// TIA Portal V20 export
FUNCTION_BLOCK "Sequence_1_WebGuid"   // FB127, LAD
TITLE = Sequence
// Sequence template programmend in ladder logic
// stored: IsIECCheckEnabled true, MemoryReserve 100, Namespace Unit1.Em3, SetENOAutomatically true
   VAR
      instSequenceLADControl { ExternalWritable := 'False'} : "LAF_ControlLadSequence";
      instSequenceLADStatus { ExternalWritable := 'False'} : "LAF_StatusLadSequence";
      statPulse { ExternalWritable := 'False'} : Array[0..999] of Bool;
      statTonTimer { ExternalWritable := 'False'} : Array[0..1099] of TON_TIME;
   END_VAR
   VAR_TEMP
      tempCustomerAction : Bool;   // Placeholder for possible actions
      tempDo_nothing_and_wait_for_init : Bool;   // Placeholder for doing nothing
      tempSafeStateCondition : Bool;   // Temp Condition for the equipment module to be in a safe state
   END_VAR
   VAR CONSTANT
      STEP_IDLE : DInt := 1;   // Idle Step
      JOB_1_STEP_01 : DInt := 101;
      JOB_1_STEP_11 : DInt := 111;
      JOB_1_STEP_21 : DInt := 121;
      JOB_1_STEP_31 : DInt := 131;
      JOB_1_STEP_41 : DInt := 141;
      JOB_1_STEP_51 : DInt := 151;
      JOB_1_STEP_61 : DInt := 161;
      JOB_1_STEP_71 : DInt := 171;
      JOB_1_STEP_81 : DInt := 181;
      JOB_1_STEP_91 : DInt := 191;
      JOB_2_STEP_01 : DInt := 201;
      JOB_2_STEP_11 : DInt := 211;
      JOB_2_STEP_21 : DInt := 221;
      JOB_2_STEP_31 : DInt := 231;
      JOB_2_STEP_41 : DInt := 241;
      JOB_2_STEP_51 : DInt := 251;
      JOB_2_STEP_61 : DInt := 261;
      JOB_2_STEP_71 : DInt := 271;
      JOB_2_STEP_81 : DInt := 281;
      JOB_2_STEP_91 : DInt := 291;
      JOB_3_STEP_01 : DInt := 301;
      JOB_3_STEP_11 : DInt := 311;
      JOB_3_STEP_21 : DInt := 321;
      JOB_3_STEP_31 : DInt := 331;
      JOB_3_STEP_41 : DInt := 341;
      JOB_3_STEP_51 : DInt := 351;
      JOB_3_STEP_61 : DInt := 361;
      JOB_3_STEP_71 : DInt := 371;
      JOB_3_STEP_81 : DInt := 381;
      JOB_3_STEP_91 : DInt := 391;
      JOB_4_STEP_01 : DInt := 401;
      JOB_4_STEP_11 : DInt := 411;
      JOB_4_STEP_21 : DInt := 421;
      JOB_4_STEP_31 : DInt := 431;
      JOB_4_STEP_41 : DInt := 441;
      JOB_4_STEP_51 : DInt := 451;
      JOB_4_STEP_61 : DInt := 461;
      JOB_4_STEP_71 : DInt := 471;
      JOB_4_STEP_81 : DInt := 481;
      JOB_4_STEP_91 : DInt := 491;
      JOB_5_STEP_01 : DInt := 501;
      JOB_5_STEP_11 : DInt := 511;
      JOB_5_STEP_21 : DInt := 521;
      JOB_5_STEP_31 : DInt := 531;
      JOB_5_STEP_41 : DInt := 541;
      JOB_5_STEP_51 : DInt := 551;
      JOB_5_STEP_61 : DInt := 561;
      JOB_5_STEP_71 : DInt := 571;
      JOB_5_STEP_81 : DInt := 581;
      JOB_5_STEP_91 : DInt := 591;
      JOB_6_STEP_01 : DInt := 601;
      JOB_6_STEP_11 : DInt := 611;
      JOB_6_STEP_21 : DInt := 621;
      JOB_6_STEP_31 : DInt := 631;
      JOB_6_STEP_41 : DInt := 641;
      JOB_6_STEP_51 : DInt := 651;
      JOB_6_STEP_61 : DInt := 661;
      JOB_6_STEP_71 : DInt := 671;
      JOB_6_STEP_81 : DInt := 681;
      JOB_6_STEP_91 : DInt := 691;
      JOB_7_STEP_01 : DInt := 701;
      JOB_7_STEP_11 : DInt := 711;
      JOB_7_STEP_21 : DInt := 721;
      JOB_7_STEP_31 : DInt := 731;
      JOB_7_STEP_41 : DInt := 741;
      JOB_7_STEP_51 : DInt := 751;
      JOB_7_STEP_61 : DInt := 761;
      JOB_7_STEP_71 : DInt := 771;
      JOB_7_STEP_81 : DInt := 781;
      JOB_7_STEP_91 : DInt := 791;
      JOB_8_STEP_01 : DInt := 801;
      JOB_8_STEP_11 : DInt := 811;
      JOB_8_STEP_21 : DInt := 821;
      JOB_8_STEP_31 : DInt := 831;
      JOB_8_STEP_41 : DInt := 841;
      JOB_8_STEP_51 : DInt := 851;
      JOB_8_STEP_61 : DInt := 861;
      JOB_8_STEP_71 : DInt := 871;
      JOB_8_STEP_81 : DInt := 881;
      JOB_8_STEP_91 : DInt := 891;
      STEP_IMMEDIATE_STOP : DInt := 901;   // Step executed when an immediate stop command is triggered for the sequence (i.e. when unit is in state aborting)
      TO_DO_INSERT_ACTIONS_HERE : Bool := TRUE;   // Template : Add actions
      TO_DO_INSERT_CONDITION_FOR_TRANSITION_HERE : Bool := TRUE;   // Template : Add conditions
      SeqDelayTime : Time := T#100ms;
      SeqNoDelayTime : Time;
      TRUE : Bool := TRUE;
      FALSE : Bool := FALSE;
   END_VAR
   VAR_TEMP   // added for the SCL form of the ladder/FBD networks
      _w1 : Bool;
      _w2 : Bool;
      _w3 : Bool;
   END_VAR
BEGIN

REGION Network 1: BLOCK INFO HEADER
   // (company) / (C) Copyright (year)
   // ---------------------------------------------------------------------------------
   // Title:                             (Title of this block)
   // Comment/Function: (that is implemented in the block)
   // Library/Family:           (that the source is dedicated to)
   // Author:                        (department / person in charge / contact)
   // Target System:          (test system with FW version)
   // Engineering:              TIA Portal (SW version)
   // Restrictions:               (OB types, etc.)
   // Requirements:           (hardware, technological package, etc.)
   // ---------------------------------------------------------------------------------
   // Change log table:
   // Version          | Date             | Signature      | Expert in charge  | Changes applied ------------------------|----------------------|-------------------------|--------------------------------|-----------------------
   // 001.000.000 | yyyy-mm-dd | 0x00000000 | (name of expert) | First released version
END_REGION

REGION Network 2: DESCRIPTION
   // This is a template block provided by the Automation Framework. It can be used to create an own project.
   // The Block Info Header is prepared to put in your own data.
   // Description of the block could be added here and the docu created by Code2Docu.
END_REGION

REGION Network 3: ******************** CONTROL ********************
END_REGION

REGION Network 4: Sequence Control
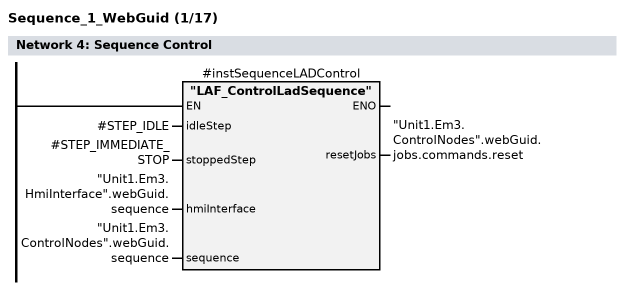
   RUNG wire#powerrail
      #instSequenceLADControl(idleStep := #STEP_IDLE, stoppedStep := #STEP_IMMEDIATE_STOP, hmiInterface := "Unit1.Em3.HmiInterface".webGuid.sequence, sequence := "Unit1.Em3.ControlNodes".webGuid.sequence, resetJobs => "Unit1.Em3.ControlNodes".webGuid.jobs.commands.reset)
   END_RUNG
   // the same network as SCL:
   #instSequenceLADControl(idleStep := #STEP_IDLE,   // "LAF_ControlLadSequence"
                           stoppedStep := #STEP_IMMEDIATE_STOP,
                           hmiInterface := "Unit1.Em3.HmiInterface".webGuid.sequence,
                           sequence := "Unit1.Em3.ControlNodes".webGuid.sequence,
                           resetJobs => "Unit1.Em3.ControlNodes".webGuid.jobs.commands.reset);
END_REGION

REGION Network 5: Step IDLE
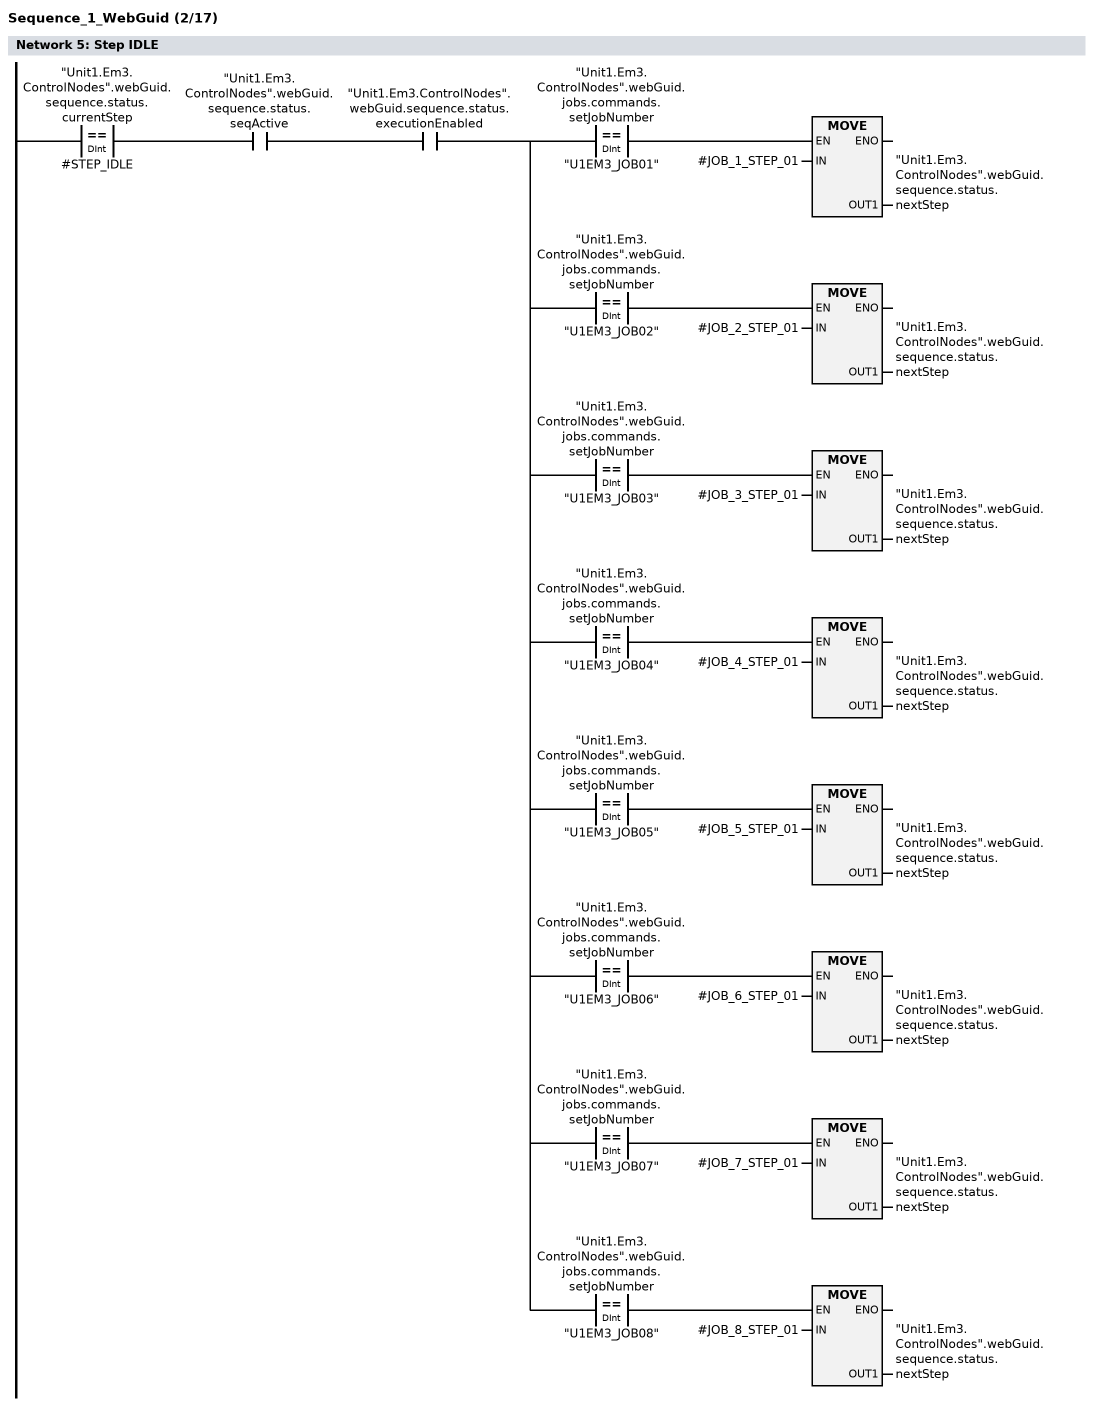
   RUNG wire#powerrail
      { S7_Templates := "SrcType := DInt" } EQ_Contact(in1 := "Unit1.Em3.ControlNodes".webGuid.sequence.status.currentStep, in2 := #STEP_IDLE)
      Contact( "Unit1.Em3.ControlNodes".webGuid.sequence.status.seqActive )
      Contact( "Unit1.Em3.ControlNodes".webGuid.sequence.status.executionEnabled )
      wire#w1
      { S7_Templates := "SrcType := DInt" } EQ_Contact(in1 := "Unit1.Em3.ControlNodes".webGuid.jobs.commands.setJobNumber, in2 := "U1EM3_JOB01")
      Move(in := #JOB_1_STEP_01, out1 => "Unit1.Em3.ControlNodes".webGuid.sequence.status.nextStep)
   END_RUNG
   RUNG wire#w1
      { S7_Templates := "SrcType := DInt" } EQ_Contact(in1 := "Unit1.Em3.ControlNodes".webGuid.jobs.commands.setJobNumber, in2 := "U1EM3_JOB02")
      Move(in := #JOB_2_STEP_01, out1 => "Unit1.Em3.ControlNodes".webGuid.sequence.status.nextStep)
   END_RUNG
   RUNG wire#w1
      { S7_Templates := "SrcType := DInt" } EQ_Contact(in1 := "Unit1.Em3.ControlNodes".webGuid.jobs.commands.setJobNumber, in2 := "U1EM3_JOB03")
      Move(in := #JOB_3_STEP_01, out1 => "Unit1.Em3.ControlNodes".webGuid.sequence.status.nextStep)
   END_RUNG
   RUNG wire#w1
      { S7_Templates := "SrcType := DInt" } EQ_Contact(in1 := "Unit1.Em3.ControlNodes".webGuid.jobs.commands.setJobNumber, in2 := "U1EM3_JOB04")
      Move(in := #JOB_4_STEP_01, out1 => "Unit1.Em3.ControlNodes".webGuid.sequence.status.nextStep)
   END_RUNG
   RUNG wire#w1
      { S7_Templates := "SrcType := DInt" } EQ_Contact(in1 := "Unit1.Em3.ControlNodes".webGuid.jobs.commands.setJobNumber, in2 := "U1EM3_JOB05")
      Move(in := #JOB_5_STEP_01, out1 => "Unit1.Em3.ControlNodes".webGuid.sequence.status.nextStep)
   END_RUNG
   RUNG wire#w1
      { S7_Templates := "SrcType := DInt" } EQ_Contact(in1 := "Unit1.Em3.ControlNodes".webGuid.jobs.commands.setJobNumber, in2 := "U1EM3_JOB06")
      Move(in := #JOB_6_STEP_01, out1 => "Unit1.Em3.ControlNodes".webGuid.sequence.status.nextStep)
   END_RUNG
   RUNG wire#w1
      { S7_Templates := "SrcType := DInt" } EQ_Contact(in1 := "Unit1.Em3.ControlNodes".webGuid.jobs.commands.setJobNumber, in2 := "U1EM3_JOB07")
      Move(in := #JOB_7_STEP_01, out1 => "Unit1.Em3.ControlNodes".webGuid.sequence.status.nextStep)
   END_RUNG
   RUNG wire#w1
      { S7_Templates := "SrcType := DInt" } EQ_Contact(in1 := "Unit1.Em3.ControlNodes".webGuid.jobs.commands.setJobNumber, in2 := "U1EM3_JOB08")
      Move(in := #JOB_8_STEP_01, out1 => "Unit1.Em3.ControlNodes".webGuid.sequence.status.nextStep)
   END_RUNG
   // the same network as SCL:
   #_w1 := ("Unit1.Em3.ControlNodes".webGuid.sequence.status.currentStep = #STEP_IDLE) AND "Unit1.Em3.ControlNodes".webGuid.sequence.status.seqActive AND "Unit1.Em3.ControlNodes".webGuid.sequence.status.executionEnabled;
   IF #_w1 AND ("Unit1.Em3.ControlNodes".webGuid.jobs.commands.setJobNumber = "U1EM3_JOB01") THEN
       "Unit1.Em3.ControlNodes".webGuid.sequence.status.nextStep := #JOB_1_STEP_01;
   END_IF;
   IF #_w1 AND ("Unit1.Em3.ControlNodes".webGuid.jobs.commands.setJobNumber = "U1EM3_JOB02") THEN
       "Unit1.Em3.ControlNodes".webGuid.sequence.status.nextStep := #JOB_2_STEP_01;
   END_IF;
   IF #_w1 AND ("Unit1.Em3.ControlNodes".webGuid.jobs.commands.setJobNumber = "U1EM3_JOB03") THEN
       "Unit1.Em3.ControlNodes".webGuid.sequence.status.nextStep := #JOB_3_STEP_01;
   END_IF;
   IF #_w1 AND ("Unit1.Em3.ControlNodes".webGuid.jobs.commands.setJobNumber = "U1EM3_JOB04") THEN
       "Unit1.Em3.ControlNodes".webGuid.sequence.status.nextStep := #JOB_4_STEP_01;
   END_IF;
   IF #_w1 AND ("Unit1.Em3.ControlNodes".webGuid.jobs.commands.setJobNumber = "U1EM3_JOB05") THEN
       "Unit1.Em3.ControlNodes".webGuid.sequence.status.nextStep := #JOB_5_STEP_01;
   END_IF;
   IF #_w1 AND ("Unit1.Em3.ControlNodes".webGuid.jobs.commands.setJobNumber = "U1EM3_JOB06") THEN
       "Unit1.Em3.ControlNodes".webGuid.sequence.status.nextStep := #JOB_6_STEP_01;
   END_IF;
   IF #_w1 AND ("Unit1.Em3.ControlNodes".webGuid.jobs.commands.setJobNumber = "U1EM3_JOB07") THEN
       "Unit1.Em3.ControlNodes".webGuid.sequence.status.nextStep := #JOB_7_STEP_01;
   END_IF;
   IF #_w1 AND ("Unit1.Em3.ControlNodes".webGuid.jobs.commands.setJobNumber = "U1EM3_JOB08") THEN
       "Unit1.Em3.ControlNodes".webGuid.sequence.status.nextStep := #JOB_8_STEP_01;
   END_IF;
END_REGION

REGION Network 6: Step IDLE Dancer WorkPos Command
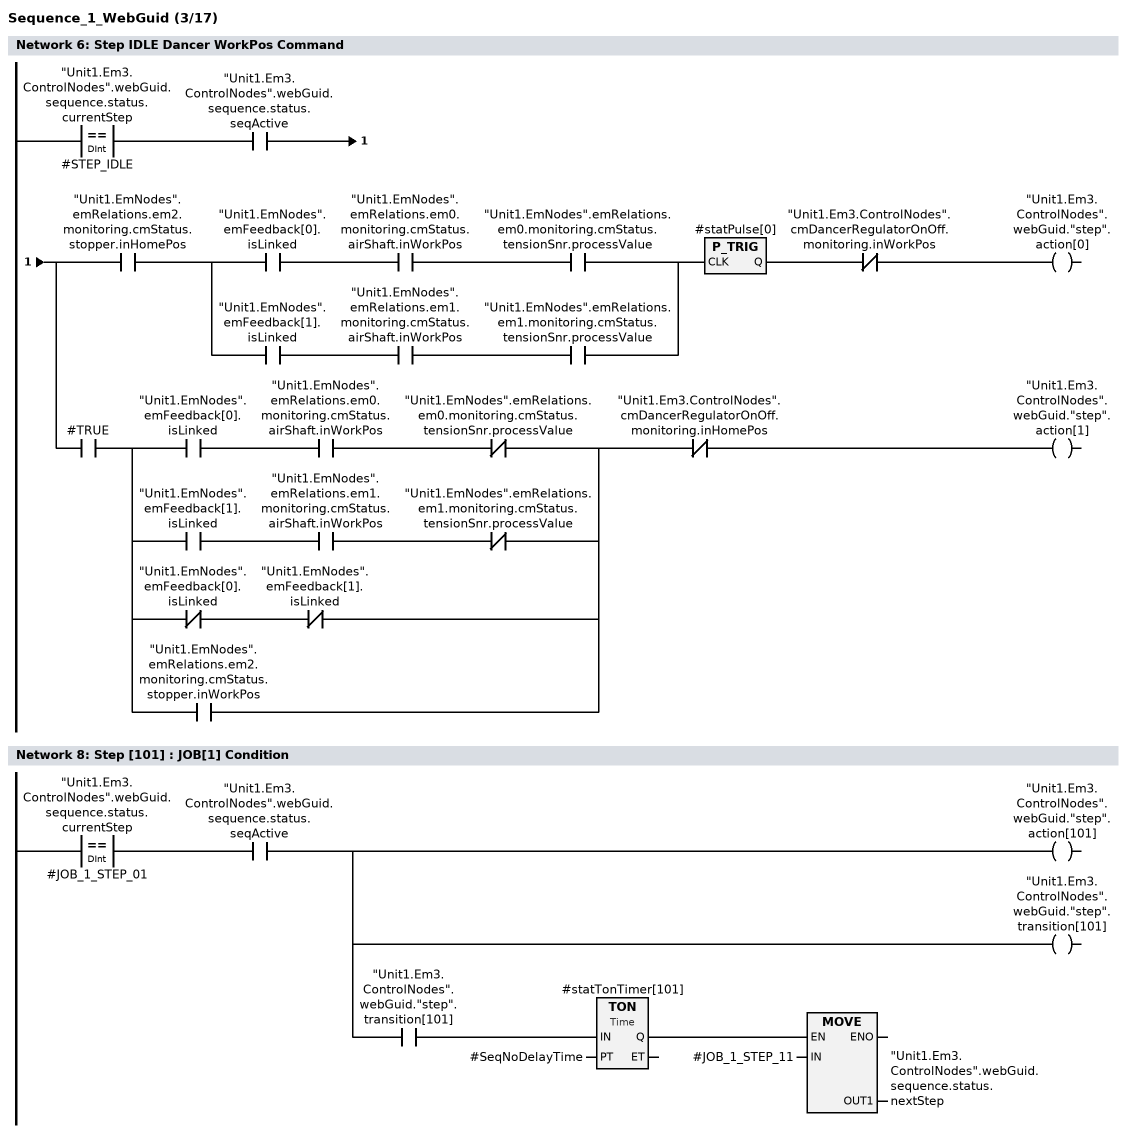
   RUNG wire#powerrail
      { S7_Templates := "SrcType := DInt" } EQ_Contact(in1 := "Unit1.Em3.ControlNodes".webGuid.sequence.status.currentStep, in2 := #STEP_IDLE)
      Contact( "Unit1.Em3.ControlNodes".webGuid.sequence.status.seqActive )
      wire#w1
      Contact( "Unit1.EmNodes".emRelations.em2.monitoring.cmStatus.stopper.inHomePos )
      wire#w2
      Contact( "Unit1.EmNodes".emFeedback[0].isLinked )
      Contact( "Unit1.EmNodes".emRelations.em0.monitoring.cmStatus.airShaft.inWorkPos )
      Contact( "Unit1.EmNodes".emRelations.em0.monitoring.cmStatus.tensionSnr.processValue )
      wire#w3
      P_Trig( #statPulse[0] )
      I_Contact( "Unit1.Em3.ControlNodes".cmDancerRegulatorOnOff.monitoring.inWorkPos )
      Coil( "Unit1.Em3.ControlNodes".webGuid."step".action[0] )
   END_RUNG
   RUNG wire#w2
      Contact( "Unit1.EmNodes".emFeedback[1].isLinked )
      Contact( "Unit1.EmNodes".emRelations.em1.monitoring.cmStatus.airShaft.inWorkPos )
      Contact( "Unit1.EmNodes".emRelations.em1.monitoring.cmStatus.tensionSnr.processValue )
   END_RUNG wire#w3
   RUNG wire#w1
      Contact( #TRUE )
      wire#w4
      Contact( "Unit1.EmNodes".emFeedback[0].isLinked )
      Contact( "Unit1.EmNodes".emRelations.em0.monitoring.cmStatus.airShaft.inWorkPos )
      I_Contact( "Unit1.EmNodes".emRelations.em0.monitoring.cmStatus.tensionSnr.processValue )
      wire#w5
      I_Contact( "Unit1.Em3.ControlNodes".cmDancerRegulatorOnOff.monitoring.inHomePos )
      Coil( "Unit1.Em3.ControlNodes".webGuid."step".action[1] )
   END_RUNG
   RUNG wire#w4
      Contact( "Unit1.EmNodes".emFeedback[1].isLinked )
      Contact( "Unit1.EmNodes".emRelations.em1.monitoring.cmStatus.airShaft.inWorkPos )
      I_Contact( "Unit1.EmNodes".emRelations.em1.monitoring.cmStatus.tensionSnr.processValue )
   END_RUNG wire#w5
   RUNG wire#w4
      I_Contact( "Unit1.EmNodes".emFeedback[0].isLinked )
      I_Contact( "Unit1.EmNodes".emFeedback[1].isLinked )
   END_RUNG wire#w5
   RUNG wire#w4
      Contact( "Unit1.EmNodes".emRelations.em2.monitoring.cmStatus.stopper.inWorkPos )
   END_RUNG wire#w5
   // the same network as SCL:
   #_w1 := ("Unit1.Em3.ControlNodes".webGuid.sequence.status.currentStep = #STEP_IDLE) AND "Unit1.Em3.ControlNodes".webGuid.sequence.status.seqActive;
   #_w2 := #_w1 AND "Unit1.EmNodes".emRelations.em2.monitoring.cmStatus.stopper.inHomePos AND (("Unit1.EmNodes".emFeedback[0].isLinked AND "Unit1.EmNodes".emRelations.em0.monitoring.cmStatus.airShaft.inWorkPos AND "Unit1.EmNodes".emRelations.em0.monitoring.cmStatus.tensionSnr.processValue) OR ("Unit1.EmNodes".emFeedback[1].isLinked AND "Unit1.EmNodes".emRelations.em1.monitoring.cmStatus.airShaft.inWorkPos AND "Unit1.EmNodes".emRelations.em1.monitoring.cmStatus.tensionSnr.processValue));
   #_w3 := #_w2 AND NOT #statPulse[0];   // rising edge
   #statPulse[0] := #_w2;
   "Unit1.Em3.ControlNodes".webGuid."step".action[0] := #_w3 AND NOT "Unit1.Em3.ControlNodes".cmDancerRegulatorOnOff.monitoring.inWorkPos;
   "Unit1.Em3.ControlNodes".webGuid."step".action[1] := #_w1 AND #TRUE AND (("Unit1.EmNodes".emFeedback[0].isLinked AND "Unit1.EmNodes".emRelations.em0.monitoring.cmStatus.airShaft.inWorkPos AND NOT "Unit1.EmNodes".emRelations.em0.monitoring.cmStatus.tensionSnr.processValue) OR ("Unit1.EmNodes".emFeedback[1].isLinked AND "Unit1.EmNodes".emRelations.em1.monitoring.cmStatus.airShaft.inWorkPos AND NOT "Unit1.EmNodes".emRelations.em1.monitoring.cmStatus.tensionSnr.processValue) OR (NOT "Unit1.EmNodes".emFeedback[0].isLinked AND NOT "Unit1.EmNodes".emFeedback[1].isLinked) OR "Unit1.EmNodes".emRelations.em2.monitoring.cmStatus.stopper.inWorkPos) AND NOT "Unit1.Em3.ControlNodes".cmDancerRegulatorOnOff.monitoring.inHomePos;
END_REGION

REGION Network 7: ******************** JOB[1] EM INITIALIZED ********************
END_REGION

REGION Network 8: Step [101] : JOB[1] Condition
   RUNG wire#powerrail
      { S7_Templates := "SrcType := DInt" } EQ_Contact(in1 := "Unit1.Em3.ControlNodes".webGuid.sequence.status.currentStep, in2 := #JOB_1_STEP_01)
      Contact( "Unit1.Em3.ControlNodes".webGuid.sequence.status.seqActive )
      wire#w1
      Coil( "Unit1.Em3.ControlNodes".webGuid."step".action[101] )
   END_RUNG
   RUNG wire#w1
      Coil( "Unit1.Em3.ControlNodes".webGuid."step".transition[101] )
   END_RUNG
   RUNG wire#w1
      Contact( "Unit1.Em3.ControlNodes".webGuid."step".transition[101] )
      { S7_Templates := "time_type := Time" } #statTonTimer[101].TON(pt := #SeqNoDelayTime, et =>)
      Move(in := #JOB_1_STEP_11, out1 => "Unit1.Em3.ControlNodes".webGuid.sequence.status.nextStep)
   END_RUNG
   // the same network as SCL:
   "Unit1.Em3.ControlNodes".webGuid."step".action[101] := ("Unit1.Em3.ControlNodes".webGuid.sequence.status.currentStep = #JOB_1_STEP_01) AND "Unit1.Em3.ControlNodes".webGuid.sequence.status.seqActive;
   "Unit1.Em3.ControlNodes".webGuid."step".transition[101] := ("Unit1.Em3.ControlNodes".webGuid.sequence.status.currentStep = #JOB_1_STEP_01) AND "Unit1.Em3.ControlNodes".webGuid.sequence.status.seqActive;
   #statTonTimer[101].TON(IN := ("Unit1.Em3.ControlNodes".webGuid.sequence.status.currentStep = #JOB_1_STEP_01) AND "Unit1.Em3.ControlNodes".webGuid.sequence.status.seqActive AND "Unit1.Em3.ControlNodes".webGuid."step".transition[101],
                          PT := #SeqNoDelayTime);
   IF #statTonTimer[101].Q THEN
       "Unit1.Em3.ControlNodes".webGuid.sequence.status.nextStep := #JOB_1_STEP_11;
   END_IF;
END_REGION

REGION Network 9: Step [111] : Web Guide EPC Mode Check
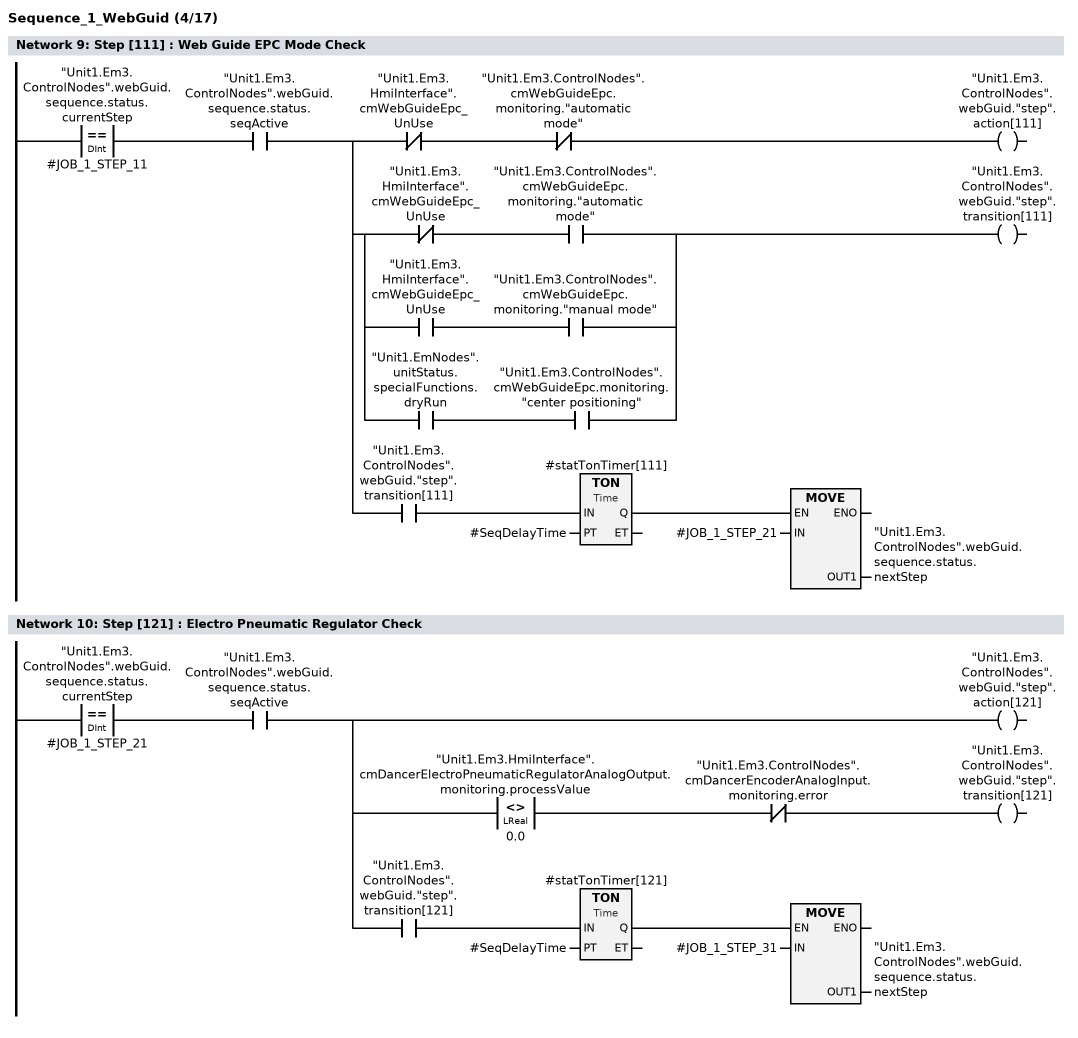
   RUNG wire#powerrail
      { S7_Templates := "SrcType := DInt" } EQ_Contact(in1 := "Unit1.Em3.ControlNodes".webGuid.sequence.status.currentStep, in2 := #JOB_1_STEP_11)
      Contact( "Unit1.Em3.ControlNodes".webGuid.sequence.status.seqActive )
      wire#w1
      I_Contact( "Unit1.Em3.HmiInterface".cmWebGuideEpc_UnUse )
      I_Contact( "Unit1.Em3.ControlNodes".cmWebGuideEpc.monitoring."automatic mode" )
      Coil( "Unit1.Em3.ControlNodes".webGuid."step".action[111] )
   END_RUNG
   RUNG wire#w1
      I_Contact( "Unit1.Em3.HmiInterface".cmWebGuideEpc_UnUse )
      Contact( "Unit1.Em3.ControlNodes".cmWebGuideEpc.monitoring."automatic mode" )
      wire#w2
      Coil( "Unit1.Em3.ControlNodes".webGuid."step".transition[111] )
   END_RUNG
   RUNG wire#w1
      Contact( "Unit1.Em3.HmiInterface".cmWebGuideEpc_UnUse )
      Contact( "Unit1.Em3.ControlNodes".cmWebGuideEpc.monitoring."manual mode" )
   END_RUNG wire#w2
   RUNG wire#w1
      Contact( "Unit1.EmNodes".unitStatus.specialFunctions.dryRun )
      Contact( "Unit1.Em3.ControlNodes".cmWebGuideEpc.monitoring."center positioning" )
   END_RUNG wire#w2
   RUNG wire#w1
      Contact( "Unit1.Em3.ControlNodes".webGuid."step".transition[111] )
      { S7_Templates := "time_type := Time" } #statTonTimer[111].TON(pt := #SeqDelayTime, et =>)
      Move(in := #JOB_1_STEP_21, out1 => "Unit1.Em3.ControlNodes".webGuid.sequence.status.nextStep)
   END_RUNG
   // the same network as SCL:
   #_w1 := ("Unit1.Em3.ControlNodes".webGuid.sequence.status.currentStep = #JOB_1_STEP_11) AND "Unit1.Em3.ControlNodes".webGuid.sequence.status.seqActive;
   "Unit1.Em3.ControlNodes".webGuid."step".action[111] := #_w1 AND NOT "Unit1.Em3.HmiInterface".cmWebGuideEpc_UnUse AND NOT "Unit1.Em3.ControlNodes".cmWebGuideEpc.monitoring."automatic mode";
   "Unit1.Em3.ControlNodes".webGuid."step".transition[111] := #_w1 AND ((NOT "Unit1.Em3.HmiInterface".cmWebGuideEpc_UnUse AND "Unit1.Em3.ControlNodes".cmWebGuideEpc.monitoring."automatic mode") OR ("Unit1.Em3.HmiInterface".cmWebGuideEpc_UnUse AND "Unit1.Em3.ControlNodes".cmWebGuideEpc.monitoring."manual mode") OR ("Unit1.EmNodes".unitStatus.specialFunctions.dryRun AND "Unit1.Em3.ControlNodes".cmWebGuideEpc.monitoring."center positioning"));
   #statTonTimer[111].TON(IN := #_w1 AND "Unit1.Em3.ControlNodes".webGuid."step".transition[111],
                          PT := #SeqDelayTime);
   IF #statTonTimer[111].Q THEN
       "Unit1.Em3.ControlNodes".webGuid.sequence.status.nextStep := #JOB_1_STEP_21;
   END_IF;
END_REGION

REGION Network 10: Step [121] : Electro Pneumatic Regulator Check
   RUNG wire#powerrail
      { S7_Templates := "SrcType := DInt" } EQ_Contact(in1 := "Unit1.Em3.ControlNodes".webGuid.sequence.status.currentStep, in2 := #JOB_1_STEP_21)
      Contact( "Unit1.Em3.ControlNodes".webGuid.sequence.status.seqActive )
      wire#w1
      Coil( "Unit1.Em3.ControlNodes".webGuid."step".action[121] )
   END_RUNG
   RUNG wire#w1
      { S7_Templates := "SrcType := LReal" } NE_Contact(in1 := "Unit1.Em3.HmiInterface".cmDancerElectroPneumaticRegulatorAnalogOutput.monitoring.processValue, in2 := 0.0)
      I_Contact( "Unit1.Em3.ControlNodes".cmDancerEncoderAnalogInput.monitoring.error )
      Coil( "Unit1.Em3.ControlNodes".webGuid."step".transition[121] )
   END_RUNG
   RUNG wire#w1
      Contact( "Unit1.Em3.ControlNodes".webGuid."step".transition[121] )
      { S7_Templates := "time_type := Time" } #statTonTimer[121].TON(pt := #SeqDelayTime, et =>)
      Move(in := #JOB_1_STEP_31, out1 => "Unit1.Em3.ControlNodes".webGuid.sequence.status.nextStep)
   END_RUNG
   // the same network as SCL:
   "Unit1.Em3.ControlNodes".webGuid."step".action[121] := ("Unit1.Em3.ControlNodes".webGuid.sequence.status.currentStep = #JOB_1_STEP_21) AND "Unit1.Em3.ControlNodes".webGuid.sequence.status.seqActive;
   "Unit1.Em3.ControlNodes".webGuid."step".transition[121] := ("Unit1.Em3.ControlNodes".webGuid.sequence.status.currentStep = #JOB_1_STEP_21) AND "Unit1.Em3.ControlNodes".webGuid.sequence.status.seqActive AND ("Unit1.Em3.HmiInterface".cmDancerElectroPneumaticRegulatorAnalogOutput.monitoring.processValue <> 0.0) AND NOT "Unit1.Em3.ControlNodes".cmDancerEncoderAnalogInput.monitoring.error;
   #statTonTimer[121].TON(IN := ("Unit1.Em3.ControlNodes".webGuid.sequence.status.currentStep = #JOB_1_STEP_21) AND "Unit1.Em3.ControlNodes".webGuid.sequence.status.seqActive AND "Unit1.Em3.ControlNodes".webGuid."step".transition[121],
                          PT := #SeqDelayTime);
   IF #statTonTimer[121].Q THEN
       "Unit1.Em3.ControlNodes".webGuid.sequence.status.nextStep := #JOB_1_STEP_31;
   END_IF;
END_REGION

REGION Network 11: Step [131] : Dancer WorkPos Command
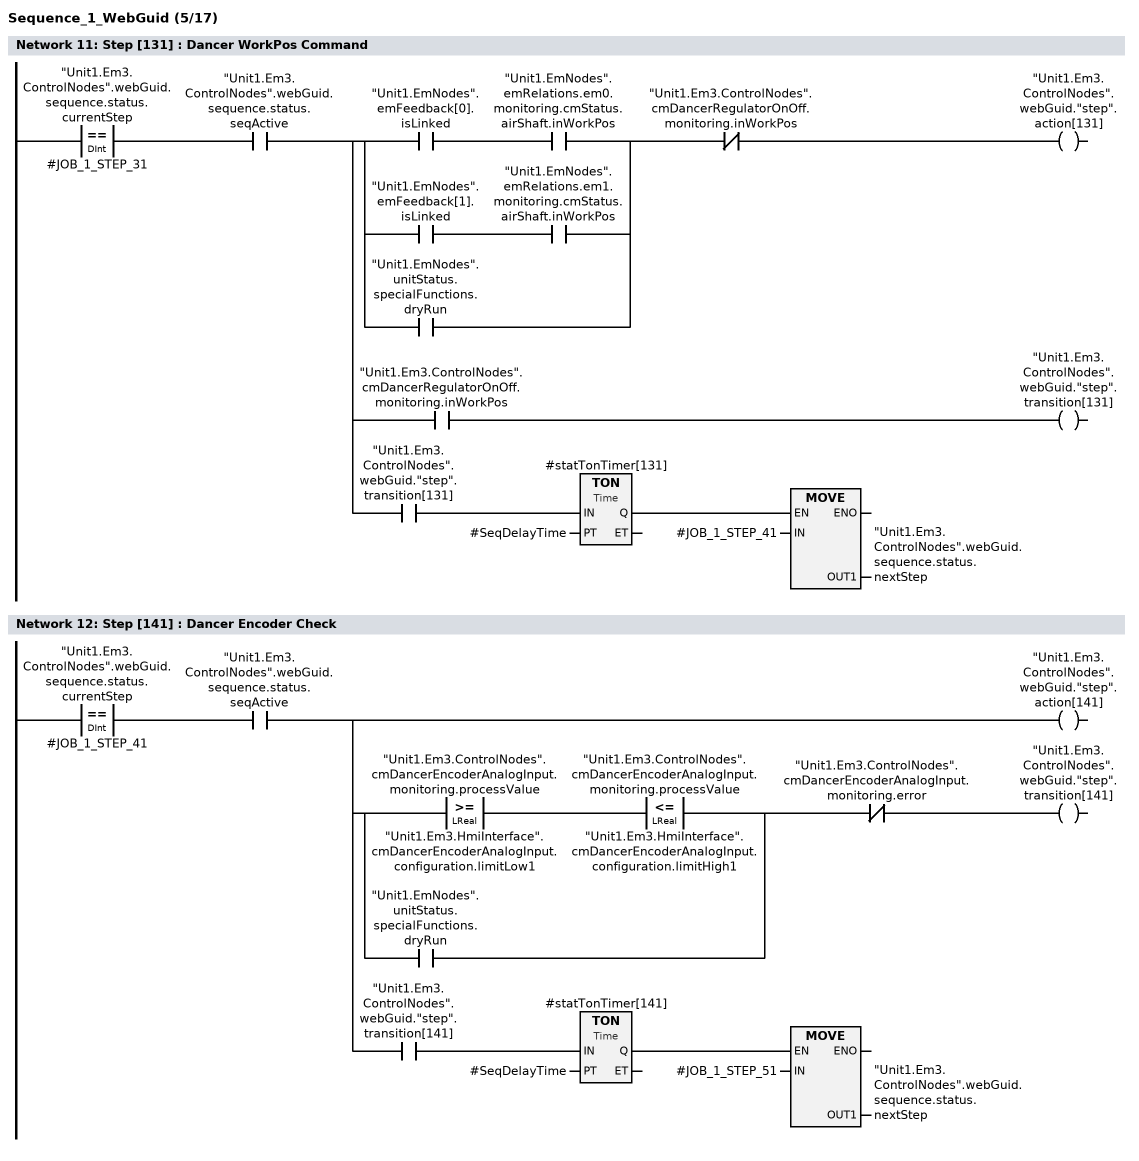
   RUNG wire#powerrail
      { S7_Templates := "SrcType := DInt" } EQ_Contact(in1 := "Unit1.Em3.ControlNodes".webGuid.sequence.status.currentStep, in2 := #JOB_1_STEP_31)
      Contact( "Unit1.Em3.ControlNodes".webGuid.sequence.status.seqActive )
      wire#w1
      Contact( "Unit1.EmNodes".emFeedback[0].isLinked )
      Contact( "Unit1.EmNodes".emRelations.em0.monitoring.cmStatus.airShaft.inWorkPos )
      wire#w2
      I_Contact( "Unit1.Em3.ControlNodes".cmDancerRegulatorOnOff.monitoring.inWorkPos )
      Coil( "Unit1.Em3.ControlNodes".webGuid."step".action[131] )
   END_RUNG
   RUNG wire#w1
      Contact( "Unit1.EmNodes".emFeedback[1].isLinked )
      Contact( "Unit1.EmNodes".emRelations.em1.monitoring.cmStatus.airShaft.inWorkPos )
   END_RUNG wire#w2
   RUNG wire#w1
      Contact( "Unit1.EmNodes".unitStatus.specialFunctions.dryRun )
   END_RUNG wire#w2
   RUNG wire#w1
      Contact( "Unit1.Em3.ControlNodes".cmDancerRegulatorOnOff.monitoring.inWorkPos )
      Coil( "Unit1.Em3.ControlNodes".webGuid."step".transition[131] )
   END_RUNG
   RUNG wire#w1
      Contact( "Unit1.Em3.ControlNodes".webGuid."step".transition[131] )
      { S7_Templates := "time_type := Time" } #statTonTimer[131].TON(pt := #SeqDelayTime, et =>)
      Move(in := #JOB_1_STEP_41, out1 => "Unit1.Em3.ControlNodes".webGuid.sequence.status.nextStep)
   END_RUNG
   // the same network as SCL:
   #_w1 := ("Unit1.Em3.ControlNodes".webGuid.sequence.status.currentStep = #JOB_1_STEP_31) AND "Unit1.Em3.ControlNodes".webGuid.sequence.status.seqActive;
   "Unit1.Em3.ControlNodes".webGuid."step".action[131] := #_w1 AND (("Unit1.EmNodes".emFeedback[0].isLinked AND "Unit1.EmNodes".emRelations.em0.monitoring.cmStatus.airShaft.inWorkPos) OR ("Unit1.EmNodes".emFeedback[1].isLinked AND "Unit1.EmNodes".emRelations.em1.monitoring.cmStatus.airShaft.inWorkPos) OR "Unit1.EmNodes".unitStatus.specialFunctions.dryRun) AND NOT "Unit1.Em3.ControlNodes".cmDancerRegulatorOnOff.monitoring.inWorkPos;
   "Unit1.Em3.ControlNodes".webGuid."step".transition[131] := #_w1 AND "Unit1.Em3.ControlNodes".cmDancerRegulatorOnOff.monitoring.inWorkPos;
   #statTonTimer[131].TON(IN := #_w1 AND "Unit1.Em3.ControlNodes".webGuid."step".transition[131],
                          PT := #SeqDelayTime);
   IF #statTonTimer[131].Q THEN
       "Unit1.Em3.ControlNodes".webGuid.sequence.status.nextStep := #JOB_1_STEP_41;
   END_IF;
END_REGION

REGION Network 12: Step [141] : Dancer Encoder Check
   RUNG wire#powerrail
      { S7_Templates := "SrcType := DInt" } EQ_Contact(in1 := "Unit1.Em3.ControlNodes".webGuid.sequence.status.currentStep, in2 := #JOB_1_STEP_41)
      Contact( "Unit1.Em3.ControlNodes".webGuid.sequence.status.seqActive )
      wire#w1
      Coil( "Unit1.Em3.ControlNodes".webGuid."step".action[141] )
   END_RUNG
   RUNG wire#w1
      { S7_Templates := "SrcType := LReal" } GE_Contact(in1 := "Unit1.Em3.ControlNodes".cmDancerEncoderAnalogInput.monitoring.processValue, in2 := "Unit1.Em3.HmiInterface".cmDancerEncoderAnalogInput.configuration.limitLow1)
      { S7_Templates := "SrcType := LReal" } LE_Contact(in1 := "Unit1.Em3.ControlNodes".cmDancerEncoderAnalogInput.monitoring.processValue, in2 := "Unit1.Em3.HmiInterface".cmDancerEncoderAnalogInput.configuration.limitHigh1)
      wire#w2
      I_Contact( "Unit1.Em3.ControlNodes".cmDancerEncoderAnalogInput.monitoring.error )
      Coil( "Unit1.Em3.ControlNodes".webGuid."step".transition[141] )
   END_RUNG
   RUNG wire#w1
      Contact( "Unit1.EmNodes".unitStatus.specialFunctions.dryRun )
   END_RUNG wire#w2
   RUNG wire#w1
      Contact( "Unit1.Em3.ControlNodes".webGuid."step".transition[141] )
      { S7_Templates := "time_type := Time" } #statTonTimer[141].TON(pt := #SeqDelayTime, et =>)
      Move(in := #JOB_1_STEP_51, out1 => "Unit1.Em3.ControlNodes".webGuid.sequence.status.nextStep)
   END_RUNG
   // the same network as SCL:
   "Unit1.Em3.ControlNodes".webGuid."step".action[141] := ("Unit1.Em3.ControlNodes".webGuid.sequence.status.currentStep = #JOB_1_STEP_41) AND "Unit1.Em3.ControlNodes".webGuid.sequence.status.seqActive;
   "Unit1.Em3.ControlNodes".webGuid."step".transition[141] := ("Unit1.Em3.ControlNodes".webGuid.sequence.status.currentStep = #JOB_1_STEP_41) AND "Unit1.Em3.ControlNodes".webGuid.sequence.status.seqActive AND ((("Unit1.Em3.ControlNodes".cmDancerEncoderAnalogInput.monitoring.processValue >= "Unit1.Em3.HmiInterface".cmDancerEncoderAnalogInput.configuration.limitLow1) AND ("Unit1.Em3.ControlNodes".cmDancerEncoderAnalogInput.monitoring.processValue <= "Unit1.Em3.HmiInterface".cmDancerEncoderAnalogInput.configuration.limitHigh1)) OR "Unit1.EmNodes".unitStatus.specialFunctions.dryRun) AND NOT "Unit1.Em3.ControlNodes".cmDancerEncoderAnalogInput.monitoring.error;
   #statTonTimer[141].TON(IN := ("Unit1.Em3.ControlNodes".webGuid.sequence.status.currentStep = #JOB_1_STEP_41) AND "Unit1.Em3.ControlNodes".webGuid.sequence.status.seqActive AND "Unit1.Em3.ControlNodes".webGuid."step".transition[141],
                          PT := #SeqDelayTime);
   IF #statTonTimer[141].Q THEN
       "Unit1.Em3.ControlNodes".webGuid.sequence.status.nextStep := #JOB_1_STEP_51;
   END_IF;
END_REGION

REGION Network 13: Step [151] : Master Virtual Axis Homed Check
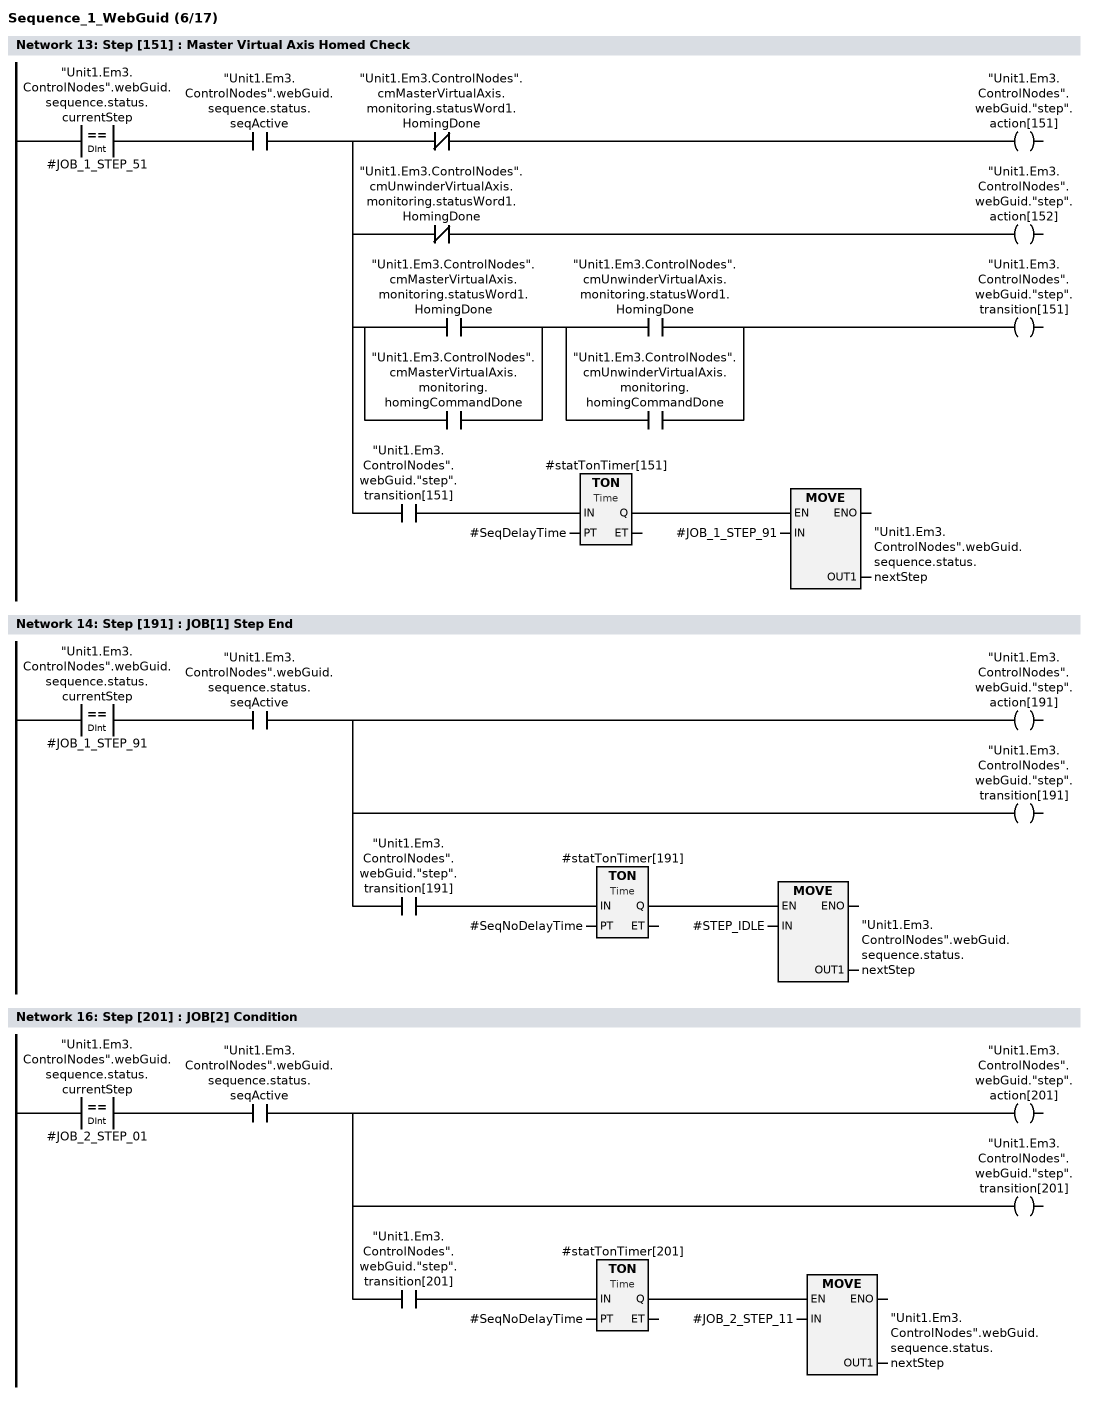
   RUNG wire#powerrail
      { S7_Templates := "SrcType := DInt" } EQ_Contact(in1 := "Unit1.Em3.ControlNodes".webGuid.sequence.status.currentStep, in2 := #JOB_1_STEP_51)
      Contact( "Unit1.Em3.ControlNodes".webGuid.sequence.status.seqActive )
      wire#w1
      I_Contact( "Unit1.Em3.ControlNodes".cmMasterVirtualAxis.monitoring.statusWord1.HomingDone )
      Coil( "Unit1.Em3.ControlNodes".webGuid."step".action[151] )
   END_RUNG
   RUNG wire#w1
      I_Contact( "Unit1.Em3.ControlNodes".cmUnwinderVirtualAxis.monitoring.statusWord1.HomingDone )
      Coil( "Unit1.Em3.ControlNodes".webGuid."step".action[152] )
   END_RUNG
   RUNG wire#w1
      Contact( "Unit1.Em3.ControlNodes".cmMasterVirtualAxis.monitoring.statusWord1.HomingDone )
      wire#w2
      Contact( "Unit1.Em3.ControlNodes".cmUnwinderVirtualAxis.monitoring.statusWord1.HomingDone )
      wire#w3
      Coil( "Unit1.Em3.ControlNodes".webGuid."step".transition[151] )
   END_RUNG
   RUNG wire#w1
      Contact( "Unit1.Em3.ControlNodes".cmMasterVirtualAxis.monitoring.homingCommandDone )
   END_RUNG wire#w2
   RUNG wire#w2
      Contact( "Unit1.Em3.ControlNodes".cmUnwinderVirtualAxis.monitoring.homingCommandDone )
   END_RUNG wire#w3
   RUNG wire#w1
      Contact( "Unit1.Em3.ControlNodes".webGuid."step".transition[151] )
      { S7_Templates := "time_type := Time" } #statTonTimer[151].TON(pt := #SeqDelayTime, et =>)
      Move(in := #JOB_1_STEP_91, out1 => "Unit1.Em3.ControlNodes".webGuid.sequence.status.nextStep)
   END_RUNG
   // the same network as SCL:
   #_w1 := ("Unit1.Em3.ControlNodes".webGuid.sequence.status.currentStep = #JOB_1_STEP_51) AND "Unit1.Em3.ControlNodes".webGuid.sequence.status.seqActive;
   "Unit1.Em3.ControlNodes".webGuid."step".action[151] := #_w1 AND NOT "Unit1.Em3.ControlNodes".cmMasterVirtualAxis.monitoring.statusWord1.HomingDone;
   "Unit1.Em3.ControlNodes".webGuid."step".action[152] := #_w1 AND NOT "Unit1.Em3.ControlNodes".cmUnwinderVirtualAxis.monitoring.statusWord1.HomingDone;
   "Unit1.Em3.ControlNodes".webGuid."step".transition[151] := #_w1 AND ("Unit1.Em3.ControlNodes".cmMasterVirtualAxis.monitoring.statusWord1.HomingDone OR "Unit1.Em3.ControlNodes".cmMasterVirtualAxis.monitoring.homingCommandDone) AND ("Unit1.Em3.ControlNodes".cmUnwinderVirtualAxis.monitoring.statusWord1.HomingDone OR "Unit1.Em3.ControlNodes".cmUnwinderVirtualAxis.monitoring.homingCommandDone);
   #statTonTimer[151].TON(IN := #_w1 AND "Unit1.Em3.ControlNodes".webGuid."step".transition[151],
                          PT := #SeqDelayTime);
   IF #statTonTimer[151].Q THEN
       "Unit1.Em3.ControlNodes".webGuid.sequence.status.nextStep := #JOB_1_STEP_91;
   END_IF;
END_REGION

REGION Network 14: Step [191] : JOB[1] Step End
   RUNG wire#powerrail
      { S7_Templates := "SrcType := DInt" } EQ_Contact(in1 := "Unit1.Em3.ControlNodes".webGuid.sequence.status.currentStep, in2 := #JOB_1_STEP_91)
      Contact( "Unit1.Em3.ControlNodes".webGuid.sequence.status.seqActive )
      wire#w1
      Coil( "Unit1.Em3.ControlNodes".webGuid."step".action[191] )
   END_RUNG
   RUNG wire#w1
      Coil( "Unit1.Em3.ControlNodes".webGuid."step".transition[191] )
   END_RUNG
   RUNG wire#w1
      Contact( "Unit1.Em3.ControlNodes".webGuid."step".transition[191] )
      { S7_Templates := "time_type := Time" } #statTonTimer[191].TON(pt := #SeqNoDelayTime, et =>)
      Move(in := #STEP_IDLE, out1 => "Unit1.Em3.ControlNodes".webGuid.sequence.status.nextStep)
   END_RUNG
   // the same network as SCL:
   "Unit1.Em3.ControlNodes".webGuid."step".action[191] := ("Unit1.Em3.ControlNodes".webGuid.sequence.status.currentStep = #JOB_1_STEP_91) AND "Unit1.Em3.ControlNodes".webGuid.sequence.status.seqActive;
   "Unit1.Em3.ControlNodes".webGuid."step".transition[191] := ("Unit1.Em3.ControlNodes".webGuid.sequence.status.currentStep = #JOB_1_STEP_91) AND "Unit1.Em3.ControlNodes".webGuid.sequence.status.seqActive;
   #statTonTimer[191].TON(IN := ("Unit1.Em3.ControlNodes".webGuid.sequence.status.currentStep = #JOB_1_STEP_91) AND "Unit1.Em3.ControlNodes".webGuid.sequence.status.seqActive AND "Unit1.Em3.ControlNodes".webGuid."step".transition[191],
                          PT := #SeqNoDelayTime);
   IF #statTonTimer[191].Q THEN
       "Unit1.Em3.ControlNodes".webGuid.sequence.status.nextStep := #STEP_IDLE;
   END_IF;
END_REGION

REGION Network 15: ******************** JOB[2] MOTION CALCULATE ********************
END_REGION

REGION Network 16: Step [201] : JOB[2] Condition
   RUNG wire#powerrail
      { S7_Templates := "SrcType := DInt" } EQ_Contact(in1 := "Unit1.Em3.ControlNodes".webGuid.sequence.status.currentStep, in2 := #JOB_2_STEP_01)
      Contact( "Unit1.Em3.ControlNodes".webGuid.sequence.status.seqActive )
      wire#w1
      Coil( "Unit1.Em3.ControlNodes".webGuid."step".action[201] )
   END_RUNG
   RUNG wire#w1
      Coil( "Unit1.Em3.ControlNodes".webGuid."step".transition[201] )
   END_RUNG
   RUNG wire#w1
      Contact( "Unit1.Em3.ControlNodes".webGuid."step".transition[201] )
      { S7_Templates := "time_type := Time" } #statTonTimer[201].TON(pt := #SeqNoDelayTime, et =>)
      Move(in := #JOB_2_STEP_11, out1 => "Unit1.Em3.ControlNodes".webGuid.sequence.status.nextStep)
   END_RUNG
   // the same network as SCL:
   "Unit1.Em3.ControlNodes".webGuid."step".action[201] := ("Unit1.Em3.ControlNodes".webGuid.sequence.status.currentStep = #JOB_2_STEP_01) AND "Unit1.Em3.ControlNodes".webGuid.sequence.status.seqActive;
   "Unit1.Em3.ControlNodes".webGuid."step".transition[201] := ("Unit1.Em3.ControlNodes".webGuid.sequence.status.currentStep = #JOB_2_STEP_01) AND "Unit1.Em3.ControlNodes".webGuid.sequence.status.seqActive;
   #statTonTimer[201].TON(IN := ("Unit1.Em3.ControlNodes".webGuid.sequence.status.currentStep = #JOB_2_STEP_01) AND "Unit1.Em3.ControlNodes".webGuid.sequence.status.seqActive AND "Unit1.Em3.ControlNodes".webGuid."step".transition[201],
                          PT := #SeqNoDelayTime);
   IF #statTonTimer[201].Q THEN
       "Unit1.Em3.ControlNodes".webGuid.sequence.status.nextStep := #JOB_2_STEP_11;
   END_IF;
END_REGION

REGION Network 17: Step [211] : ReelCutMain Stop Command
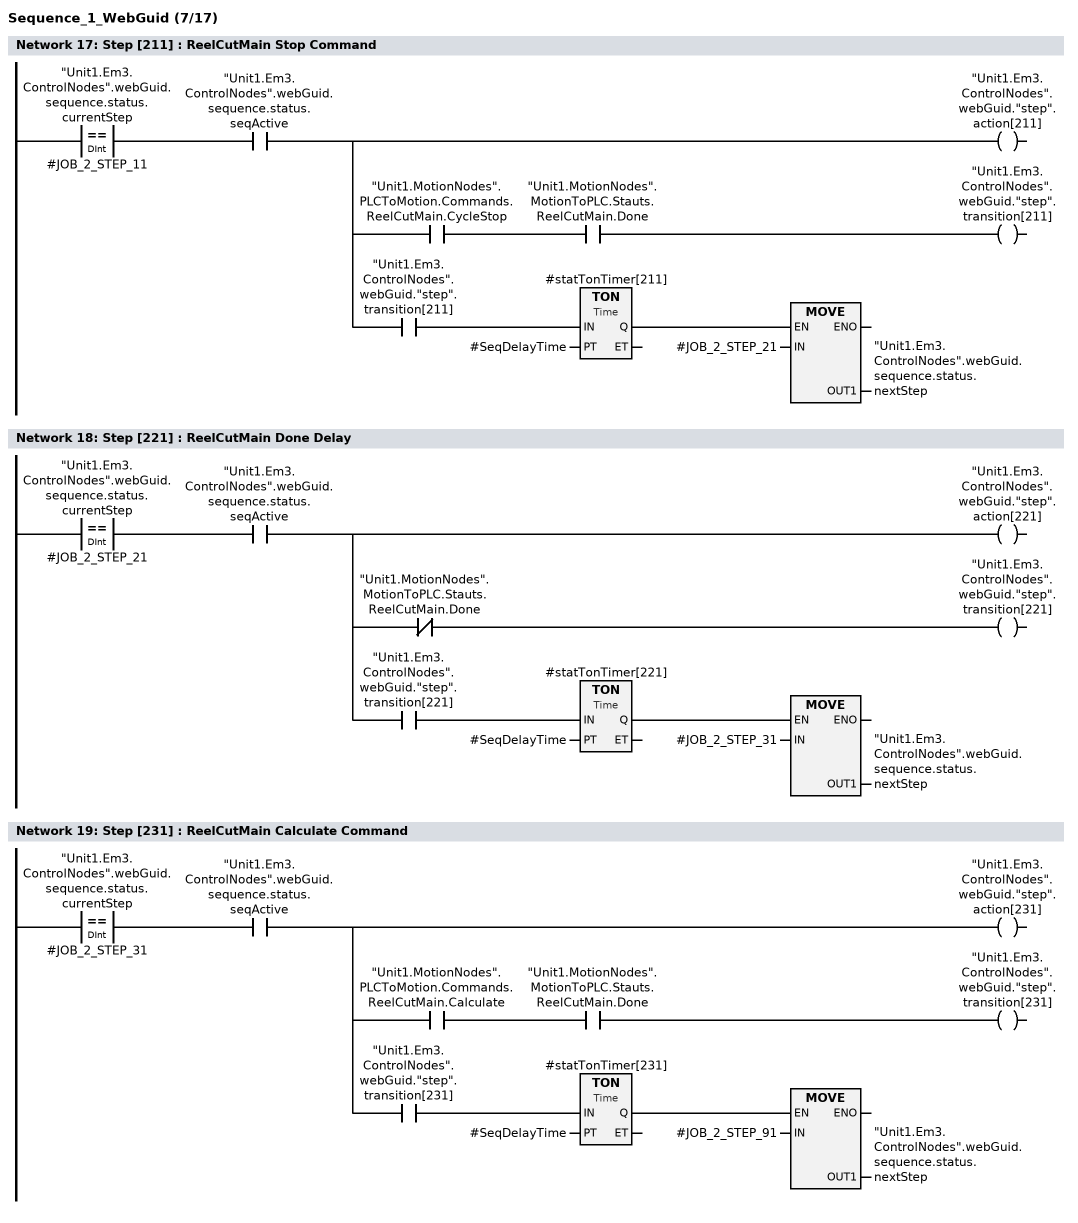
   RUNG wire#powerrail
      { S7_Templates := "SrcType := DInt" } EQ_Contact(in1 := "Unit1.Em3.ControlNodes".webGuid.sequence.status.currentStep, in2 := #JOB_2_STEP_11)
      Contact( "Unit1.Em3.ControlNodes".webGuid.sequence.status.seqActive )
      wire#w1
      Coil( "Unit1.Em3.ControlNodes".webGuid."step".action[211] )
   END_RUNG
   RUNG wire#w1
      Contact( "Unit1.MotionNodes".PLCToMotion.Commands.ReelCutMain.CycleStop )
      Contact( "Unit1.MotionNodes".MotionToPLC.Stauts.ReelCutMain.Done )
      Coil( "Unit1.Em3.ControlNodes".webGuid."step".transition[211] )
   END_RUNG
   RUNG wire#w1
      Contact( "Unit1.Em3.ControlNodes".webGuid."step".transition[211] )
      { S7_Templates := "time_type := Time" } #statTonTimer[211].TON(pt := #SeqDelayTime, et =>)
      Move(in := #JOB_2_STEP_21, out1 => "Unit1.Em3.ControlNodes".webGuid.sequence.status.nextStep)
   END_RUNG
   // the same network as SCL:
   "Unit1.Em3.ControlNodes".webGuid."step".action[211] := ("Unit1.Em3.ControlNodes".webGuid.sequence.status.currentStep = #JOB_2_STEP_11) AND "Unit1.Em3.ControlNodes".webGuid.sequence.status.seqActive;
   "Unit1.Em3.ControlNodes".webGuid."step".transition[211] := ("Unit1.Em3.ControlNodes".webGuid.sequence.status.currentStep = #JOB_2_STEP_11) AND "Unit1.Em3.ControlNodes".webGuid.sequence.status.seqActive AND "Unit1.MotionNodes".PLCToMotion.Commands.ReelCutMain.CycleStop AND "Unit1.MotionNodes".MotionToPLC.Stauts.ReelCutMain.Done;
   #statTonTimer[211].TON(IN := ("Unit1.Em3.ControlNodes".webGuid.sequence.status.currentStep = #JOB_2_STEP_11) AND "Unit1.Em3.ControlNodes".webGuid.sequence.status.seqActive AND "Unit1.Em3.ControlNodes".webGuid."step".transition[211],
                          PT := #SeqDelayTime);
   IF #statTonTimer[211].Q THEN
       "Unit1.Em3.ControlNodes".webGuid.sequence.status.nextStep := #JOB_2_STEP_21;
   END_IF;
END_REGION

REGION Network 18: Step [221] : ReelCutMain Done Delay
   RUNG wire#powerrail
      { S7_Templates := "SrcType := DInt" } EQ_Contact(in1 := "Unit1.Em3.ControlNodes".webGuid.sequence.status.currentStep, in2 := #JOB_2_STEP_21)
      Contact( "Unit1.Em3.ControlNodes".webGuid.sequence.status.seqActive )
      wire#w1
      Coil( "Unit1.Em3.ControlNodes".webGuid."step".action[221] )
   END_RUNG
   RUNG wire#w1
      I_Contact( "Unit1.MotionNodes".MotionToPLC.Stauts.ReelCutMain.Done )
      Coil( "Unit1.Em3.ControlNodes".webGuid."step".transition[221] )
   END_RUNG
   RUNG wire#w1
      Contact( "Unit1.Em3.ControlNodes".webGuid."step".transition[221] )
      { S7_Templates := "time_type := Time" } #statTonTimer[221].TON(pt := #SeqDelayTime, et =>)
      Move(in := #JOB_2_STEP_31, out1 => "Unit1.Em3.ControlNodes".webGuid.sequence.status.nextStep)
   END_RUNG
   // the same network as SCL:
   "Unit1.Em3.ControlNodes".webGuid."step".action[221] := ("Unit1.Em3.ControlNodes".webGuid.sequence.status.currentStep = #JOB_2_STEP_21) AND "Unit1.Em3.ControlNodes".webGuid.sequence.status.seqActive;
   "Unit1.Em3.ControlNodes".webGuid."step".transition[221] := ("Unit1.Em3.ControlNodes".webGuid.sequence.status.currentStep = #JOB_2_STEP_21) AND "Unit1.Em3.ControlNodes".webGuid.sequence.status.seqActive AND NOT "Unit1.MotionNodes".MotionToPLC.Stauts.ReelCutMain.Done;
   #statTonTimer[221].TON(IN := ("Unit1.Em3.ControlNodes".webGuid.sequence.status.currentStep = #JOB_2_STEP_21) AND "Unit1.Em3.ControlNodes".webGuid.sequence.status.seqActive AND "Unit1.Em3.ControlNodes".webGuid."step".transition[221],
                          PT := #SeqDelayTime);
   IF #statTonTimer[221].Q THEN
       "Unit1.Em3.ControlNodes".webGuid.sequence.status.nextStep := #JOB_2_STEP_31;
   END_IF;
END_REGION

REGION Network 19: Step [231] : ReelCutMain Calculate Command
   RUNG wire#powerrail
      { S7_Templates := "SrcType := DInt" } EQ_Contact(in1 := "Unit1.Em3.ControlNodes".webGuid.sequence.status.currentStep, in2 := #JOB_2_STEP_31)
      Contact( "Unit1.Em3.ControlNodes".webGuid.sequence.status.seqActive )
      wire#w1
      Coil( "Unit1.Em3.ControlNodes".webGuid."step".action[231] )
   END_RUNG
   RUNG wire#w1
      Contact( "Unit1.MotionNodes".PLCToMotion.Commands.ReelCutMain.Calculate )
      Contact( "Unit1.MotionNodes".MotionToPLC.Stauts.ReelCutMain.Done )
      Coil( "Unit1.Em3.ControlNodes".webGuid."step".transition[231] )
   END_RUNG
   RUNG wire#w1
      Contact( "Unit1.Em3.ControlNodes".webGuid."step".transition[231] )
      { S7_Templates := "time_type := Time" } #statTonTimer[231].TON(pt := #SeqDelayTime, et =>)
      Move(in := #JOB_2_STEP_91, out1 => "Unit1.Em3.ControlNodes".webGuid.sequence.status.nextStep)
   END_RUNG
   // the same network as SCL:
   "Unit1.Em3.ControlNodes".webGuid."step".action[231] := ("Unit1.Em3.ControlNodes".webGuid.sequence.status.currentStep = #JOB_2_STEP_31) AND "Unit1.Em3.ControlNodes".webGuid.sequence.status.seqActive;
   "Unit1.Em3.ControlNodes".webGuid."step".transition[231] := ("Unit1.Em3.ControlNodes".webGuid.sequence.status.currentStep = #JOB_2_STEP_31) AND "Unit1.Em3.ControlNodes".webGuid.sequence.status.seqActive AND "Unit1.MotionNodes".PLCToMotion.Commands.ReelCutMain.Calculate AND "Unit1.MotionNodes".MotionToPLC.Stauts.ReelCutMain.Done;
   #statTonTimer[231].TON(IN := ("Unit1.Em3.ControlNodes".webGuid.sequence.status.currentStep = #JOB_2_STEP_31) AND "Unit1.Em3.ControlNodes".webGuid.sequence.status.seqActive AND "Unit1.Em3.ControlNodes".webGuid."step".transition[231],
                          PT := #SeqDelayTime);
   IF #statTonTimer[231].Q THEN
       "Unit1.Em3.ControlNodes".webGuid.sequence.status.nextStep := #JOB_2_STEP_91;
   END_IF;
END_REGION

REGION Network 20: Step [291] : JOB[2] Step End
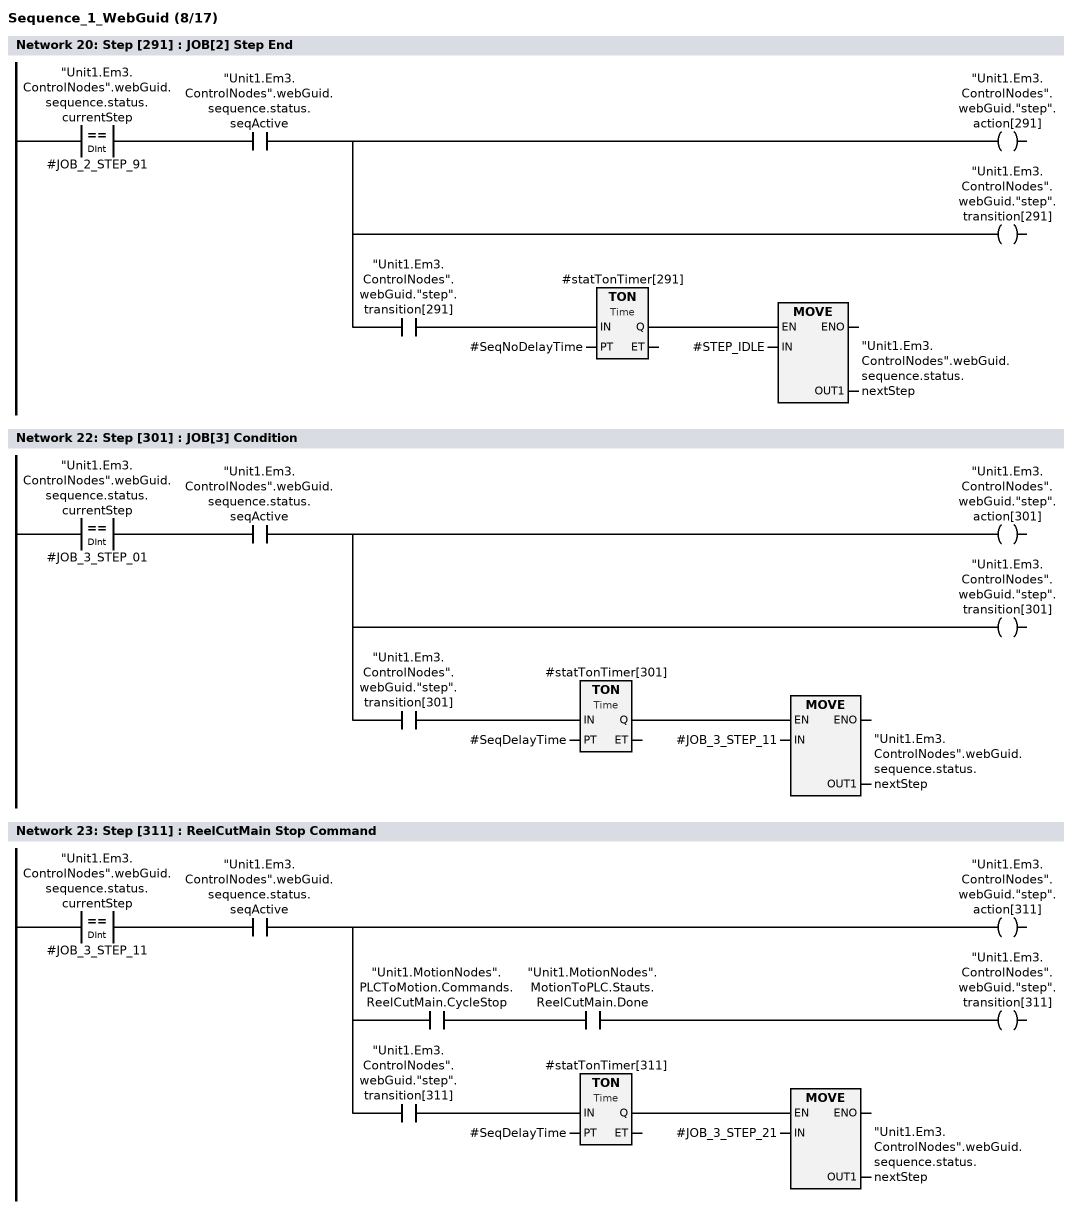
   RUNG wire#powerrail
      { S7_Templates := "SrcType := DInt" } EQ_Contact(in1 := "Unit1.Em3.ControlNodes".webGuid.sequence.status.currentStep, in2 := #JOB_2_STEP_91)
      Contact( "Unit1.Em3.ControlNodes".webGuid.sequence.status.seqActive )
      wire#w1
      Coil( "Unit1.Em3.ControlNodes".webGuid."step".action[291] )
   END_RUNG
   RUNG wire#w1
      Coil( "Unit1.Em3.ControlNodes".webGuid."step".transition[291] )
   END_RUNG
   RUNG wire#w1
      Contact( "Unit1.Em3.ControlNodes".webGuid."step".transition[291] )
      { S7_Templates := "time_type := Time" } #statTonTimer[291].TON(pt := #SeqNoDelayTime, et =>)
      Move(in := #STEP_IDLE, out1 => "Unit1.Em3.ControlNodes".webGuid.sequence.status.nextStep)
   END_RUNG
   // the same network as SCL:
   "Unit1.Em3.ControlNodes".webGuid."step".action[291] := ("Unit1.Em3.ControlNodes".webGuid.sequence.status.currentStep = #JOB_2_STEP_91) AND "Unit1.Em3.ControlNodes".webGuid.sequence.status.seqActive;
   "Unit1.Em3.ControlNodes".webGuid."step".transition[291] := ("Unit1.Em3.ControlNodes".webGuid.sequence.status.currentStep = #JOB_2_STEP_91) AND "Unit1.Em3.ControlNodes".webGuid.sequence.status.seqActive;
   #statTonTimer[291].TON(IN := ("Unit1.Em3.ControlNodes".webGuid.sequence.status.currentStep = #JOB_2_STEP_91) AND "Unit1.Em3.ControlNodes".webGuid.sequence.status.seqActive AND "Unit1.Em3.ControlNodes".webGuid."step".transition[291],
                          PT := #SeqNoDelayTime);
   IF #statTonTimer[291].Q THEN
       "Unit1.Em3.ControlNodes".webGuid.sequence.status.nextStep := #STEP_IDLE;
   END_IF;
END_REGION

REGION Network 21: ******************** JOB[3] MOTION ONE CELL ********************
END_REGION

REGION Network 22: Step [301] : JOB[3] Condition
   RUNG wire#powerrail
      { S7_Templates := "SrcType := DInt" } EQ_Contact(in1 := "Unit1.Em3.ControlNodes".webGuid.sequence.status.currentStep, in2 := #JOB_3_STEP_01)
      Contact( "Unit1.Em3.ControlNodes".webGuid.sequence.status.seqActive )
      wire#w1
      Coil( "Unit1.Em3.ControlNodes".webGuid."step".action[301] )
   END_RUNG
   RUNG wire#w1
      Coil( "Unit1.Em3.ControlNodes".webGuid."step".transition[301] )
   END_RUNG
   RUNG wire#w1
      Contact( "Unit1.Em3.ControlNodes".webGuid."step".transition[301] )
      { S7_Templates := "time_type := Time" } #statTonTimer[301].TON(pt := #SeqDelayTime, et =>)
      Move(in := #JOB_3_STEP_11, out1 => "Unit1.Em3.ControlNodes".webGuid.sequence.status.nextStep)
   END_RUNG
   // the same network as SCL:
   "Unit1.Em3.ControlNodes".webGuid."step".action[301] := ("Unit1.Em3.ControlNodes".webGuid.sequence.status.currentStep = #JOB_3_STEP_01) AND "Unit1.Em3.ControlNodes".webGuid.sequence.status.seqActive;
   "Unit1.Em3.ControlNodes".webGuid."step".transition[301] := ("Unit1.Em3.ControlNodes".webGuid.sequence.status.currentStep = #JOB_3_STEP_01) AND "Unit1.Em3.ControlNodes".webGuid.sequence.status.seqActive;
   #statTonTimer[301].TON(IN := ("Unit1.Em3.ControlNodes".webGuid.sequence.status.currentStep = #JOB_3_STEP_01) AND "Unit1.Em3.ControlNodes".webGuid.sequence.status.seqActive AND "Unit1.Em3.ControlNodes".webGuid."step".transition[301],
                          PT := #SeqDelayTime);
   IF #statTonTimer[301].Q THEN
       "Unit1.Em3.ControlNodes".webGuid.sequence.status.nextStep := #JOB_3_STEP_11;
   END_IF;
END_REGION

REGION Network 23: Step [311] : ReelCutMain Stop Command
   RUNG wire#powerrail
      { S7_Templates := "SrcType := DInt" } EQ_Contact(in1 := "Unit1.Em3.ControlNodes".webGuid.sequence.status.currentStep, in2 := #JOB_3_STEP_11)
      Contact( "Unit1.Em3.ControlNodes".webGuid.sequence.status.seqActive )
      wire#w1
      Coil( "Unit1.Em3.ControlNodes".webGuid."step".action[311] )
   END_RUNG
   RUNG wire#w1
      Contact( "Unit1.MotionNodes".PLCToMotion.Commands.ReelCutMain.CycleStop )
      Contact( "Unit1.MotionNodes".MotionToPLC.Stauts.ReelCutMain.Done )
      Coil( "Unit1.Em3.ControlNodes".webGuid."step".transition[311] )
   END_RUNG
   RUNG wire#w1
      Contact( "Unit1.Em3.ControlNodes".webGuid."step".transition[311] )
      { S7_Templates := "time_type := Time" } #statTonTimer[311].TON(pt := #SeqDelayTime, et =>)
      Move(in := #JOB_3_STEP_21, out1 => "Unit1.Em3.ControlNodes".webGuid.sequence.status.nextStep)
   END_RUNG
   // the same network as SCL:
   "Unit1.Em3.ControlNodes".webGuid."step".action[311] := ("Unit1.Em3.ControlNodes".webGuid.sequence.status.currentStep = #JOB_3_STEP_11) AND "Unit1.Em3.ControlNodes".webGuid.sequence.status.seqActive;
   "Unit1.Em3.ControlNodes".webGuid."step".transition[311] := ("Unit1.Em3.ControlNodes".webGuid.sequence.status.currentStep = #JOB_3_STEP_11) AND "Unit1.Em3.ControlNodes".webGuid.sequence.status.seqActive AND "Unit1.MotionNodes".PLCToMotion.Commands.ReelCutMain.CycleStop AND "Unit1.MotionNodes".MotionToPLC.Stauts.ReelCutMain.Done;
   #statTonTimer[311].TON(IN := ("Unit1.Em3.ControlNodes".webGuid.sequence.status.currentStep = #JOB_3_STEP_11) AND "Unit1.Em3.ControlNodes".webGuid.sequence.status.seqActive AND "Unit1.Em3.ControlNodes".webGuid."step".transition[311],
                          PT := #SeqDelayTime);
   IF #statTonTimer[311].Q THEN
       "Unit1.Em3.ControlNodes".webGuid.sequence.status.nextStep := #JOB_3_STEP_21;
   END_IF;
END_REGION

REGION Network 24: Step [321] : ReelCutMain Done Delay
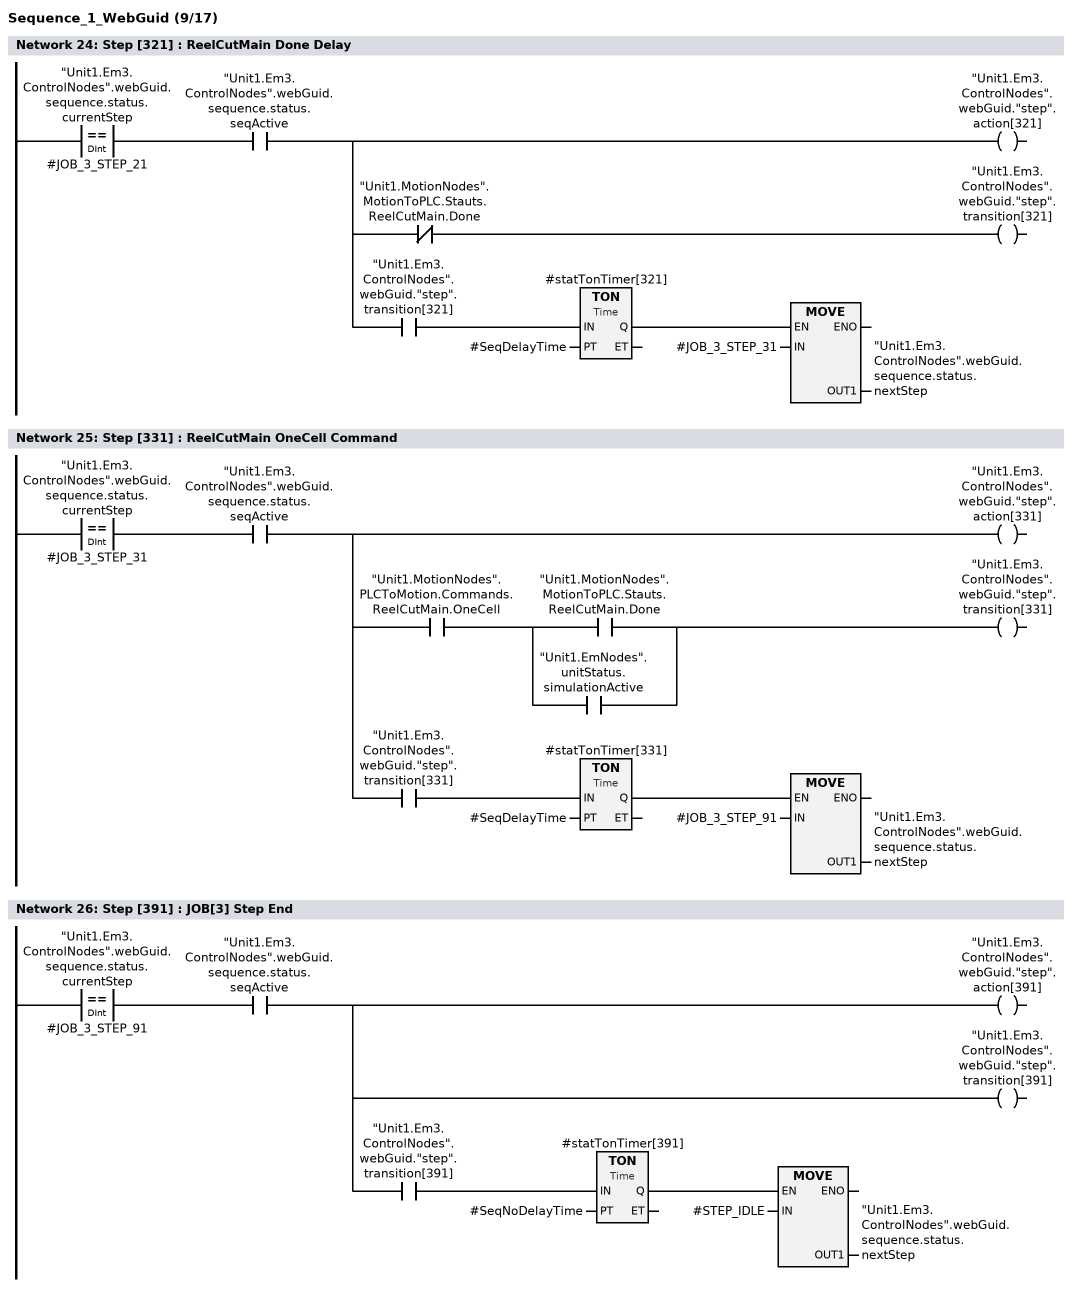
   RUNG wire#powerrail
      { S7_Templates := "SrcType := DInt" } EQ_Contact(in1 := "Unit1.Em3.ControlNodes".webGuid.sequence.status.currentStep, in2 := #JOB_3_STEP_21)
      Contact( "Unit1.Em3.ControlNodes".webGuid.sequence.status.seqActive )
      wire#w1
      Coil( "Unit1.Em3.ControlNodes".webGuid."step".action[321] )
   END_RUNG
   RUNG wire#w1
      I_Contact( "Unit1.MotionNodes".MotionToPLC.Stauts.ReelCutMain.Done )
      Coil( "Unit1.Em3.ControlNodes".webGuid."step".transition[321] )
   END_RUNG
   RUNG wire#w1
      Contact( "Unit1.Em3.ControlNodes".webGuid."step".transition[321] )
      { S7_Templates := "time_type := Time" } #statTonTimer[321].TON(pt := #SeqDelayTime, et =>)
      Move(in := #JOB_3_STEP_31, out1 => "Unit1.Em3.ControlNodes".webGuid.sequence.status.nextStep)
   END_RUNG
   // the same network as SCL:
   "Unit1.Em3.ControlNodes".webGuid."step".action[321] := ("Unit1.Em3.ControlNodes".webGuid.sequence.status.currentStep = #JOB_3_STEP_21) AND "Unit1.Em3.ControlNodes".webGuid.sequence.status.seqActive;
   "Unit1.Em3.ControlNodes".webGuid."step".transition[321] := ("Unit1.Em3.ControlNodes".webGuid.sequence.status.currentStep = #JOB_3_STEP_21) AND "Unit1.Em3.ControlNodes".webGuid.sequence.status.seqActive AND NOT "Unit1.MotionNodes".MotionToPLC.Stauts.ReelCutMain.Done;
   #statTonTimer[321].TON(IN := ("Unit1.Em3.ControlNodes".webGuid.sequence.status.currentStep = #JOB_3_STEP_21) AND "Unit1.Em3.ControlNodes".webGuid.sequence.status.seqActive AND "Unit1.Em3.ControlNodes".webGuid."step".transition[321],
                          PT := #SeqDelayTime);
   IF #statTonTimer[321].Q THEN
       "Unit1.Em3.ControlNodes".webGuid.sequence.status.nextStep := #JOB_3_STEP_31;
   END_IF;
END_REGION

REGION Network 25: Step [331] : ReelCutMain OneCell Command
   RUNG wire#powerrail
      { S7_Templates := "SrcType := DInt" } EQ_Contact(in1 := "Unit1.Em3.ControlNodes".webGuid.sequence.status.currentStep, in2 := #JOB_3_STEP_31)
      Contact( "Unit1.Em3.ControlNodes".webGuid.sequence.status.seqActive )
      wire#w1
      Coil( "Unit1.Em3.ControlNodes".webGuid."step".action[331] )
   END_RUNG
   RUNG wire#w1
      Contact( "Unit1.MotionNodes".PLCToMotion.Commands.ReelCutMain.OneCell )
      wire#w2
      Contact( "Unit1.MotionNodes".MotionToPLC.Stauts.ReelCutMain.Done )
      wire#w3
      Coil( "Unit1.Em3.ControlNodes".webGuid."step".transition[331] )
   END_RUNG
   RUNG wire#w2
      Contact( "Unit1.EmNodes".unitStatus.simulationActive )
   END_RUNG wire#w3
   RUNG wire#w1
      Contact( "Unit1.Em3.ControlNodes".webGuid."step".transition[331] )
      { S7_Templates := "time_type := Time" } #statTonTimer[331].TON(pt := #SeqDelayTime, et =>)
      Move(in := #JOB_3_STEP_91, out1 => "Unit1.Em3.ControlNodes".webGuid.sequence.status.nextStep)
   END_RUNG
   // the same network as SCL:
   "Unit1.Em3.ControlNodes".webGuid."step".action[331] := ("Unit1.Em3.ControlNodes".webGuid.sequence.status.currentStep = #JOB_3_STEP_31) AND "Unit1.Em3.ControlNodes".webGuid.sequence.status.seqActive;
   "Unit1.Em3.ControlNodes".webGuid."step".transition[331] := ("Unit1.Em3.ControlNodes".webGuid.sequence.status.currentStep = #JOB_3_STEP_31) AND "Unit1.Em3.ControlNodes".webGuid.sequence.status.seqActive AND "Unit1.MotionNodes".PLCToMotion.Commands.ReelCutMain.OneCell AND ("Unit1.MotionNodes".MotionToPLC.Stauts.ReelCutMain.Done OR "Unit1.EmNodes".unitStatus.simulationActive);
   #statTonTimer[331].TON(IN := ("Unit1.Em3.ControlNodes".webGuid.sequence.status.currentStep = #JOB_3_STEP_31) AND "Unit1.Em3.ControlNodes".webGuid.sequence.status.seqActive AND "Unit1.Em3.ControlNodes".webGuid."step".transition[331],
                          PT := #SeqDelayTime);
   IF #statTonTimer[331].Q THEN
       "Unit1.Em3.ControlNodes".webGuid.sequence.status.nextStep := #JOB_3_STEP_91;
   END_IF;
END_REGION

REGION Network 26: Step [391] : JOB[3] Step End
   RUNG wire#powerrail
      { S7_Templates := "SrcType := DInt" } EQ_Contact(in1 := "Unit1.Em3.ControlNodes".webGuid.sequence.status.currentStep, in2 := #JOB_3_STEP_91)
      Contact( "Unit1.Em3.ControlNodes".webGuid.sequence.status.seqActive )
      wire#w1
      Coil( "Unit1.Em3.ControlNodes".webGuid."step".action[391] )
   END_RUNG
   RUNG wire#w1
      Coil( "Unit1.Em3.ControlNodes".webGuid."step".transition[391] )
   END_RUNG
   RUNG wire#w1
      Contact( "Unit1.Em3.ControlNodes".webGuid."step".transition[391] )
      { S7_Templates := "time_type := Time" } #statTonTimer[391].TON(pt := #SeqNoDelayTime, et =>)
      Move(in := #STEP_IDLE, out1 => "Unit1.Em3.ControlNodes".webGuid.sequence.status.nextStep)
   END_RUNG
   // the same network as SCL:
   "Unit1.Em3.ControlNodes".webGuid."step".action[391] := ("Unit1.Em3.ControlNodes".webGuid.sequence.status.currentStep = #JOB_3_STEP_91) AND "Unit1.Em3.ControlNodes".webGuid.sequence.status.seqActive;
   "Unit1.Em3.ControlNodes".webGuid."step".transition[391] := ("Unit1.Em3.ControlNodes".webGuid.sequence.status.currentStep = #JOB_3_STEP_91) AND "Unit1.Em3.ControlNodes".webGuid.sequence.status.seqActive;
   #statTonTimer[391].TON(IN := ("Unit1.Em3.ControlNodes".webGuid.sequence.status.currentStep = #JOB_3_STEP_91) AND "Unit1.Em3.ControlNodes".webGuid.sequence.status.seqActive AND "Unit1.Em3.ControlNodes".webGuid."step".transition[391],
                          PT := #SeqNoDelayTime);
   IF #statTonTimer[391].Q THEN
       "Unit1.Em3.ControlNodes".webGuid.sequence.status.nextStep := #STEP_IDLE;
   END_IF;
END_REGION

REGION Network 27: ******************** JOB[4] MOTION FULL STEP ********************
END_REGION

REGION Network 28: Step [401] : JOB[4] Condition
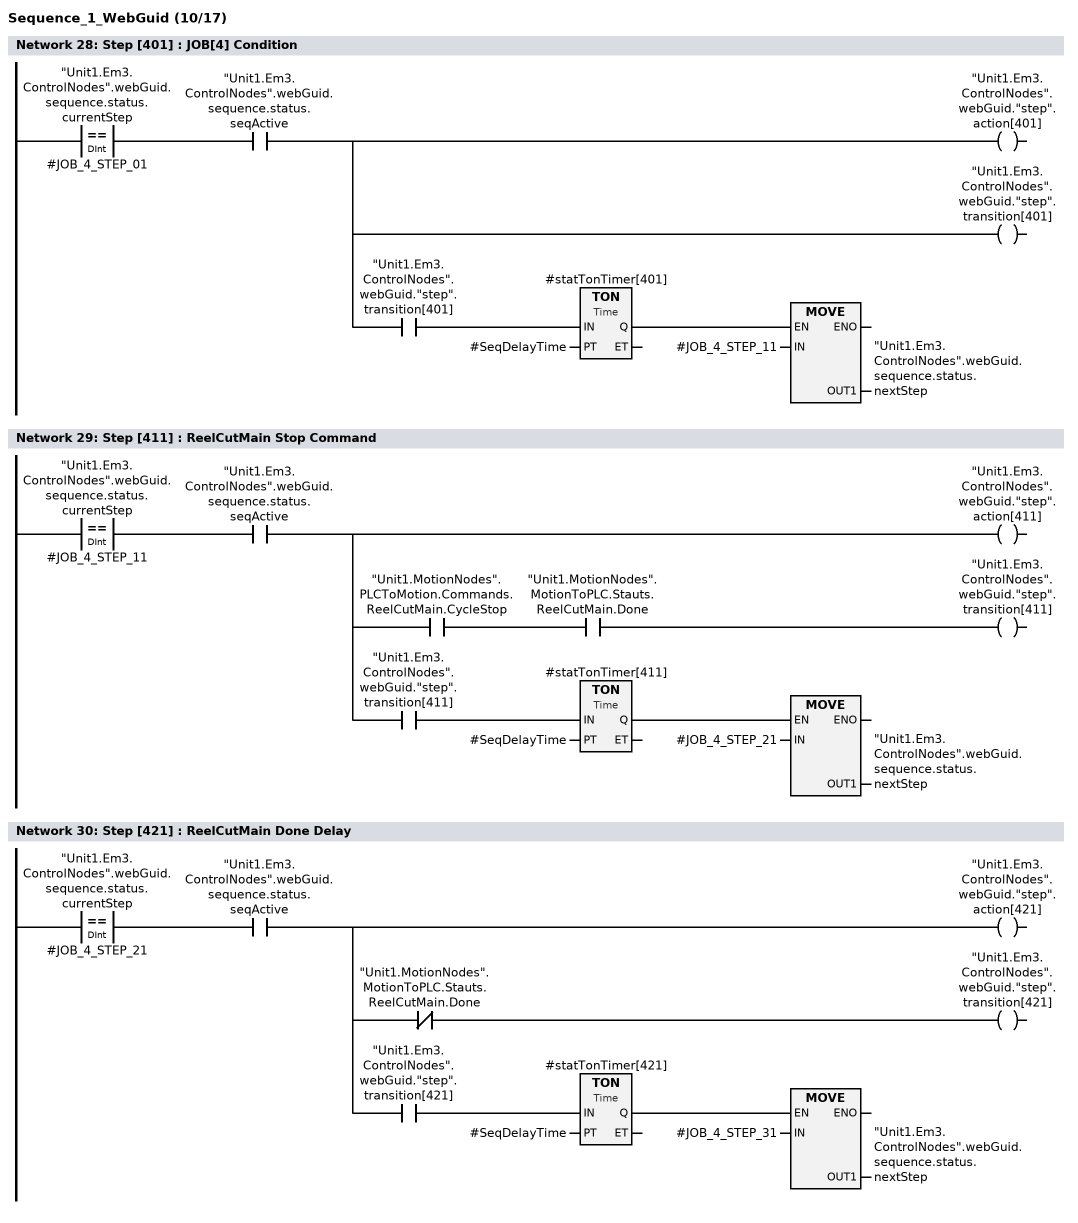
   RUNG wire#powerrail
      { S7_Templates := "SrcType := DInt" } EQ_Contact(in1 := "Unit1.Em3.ControlNodes".webGuid.sequence.status.currentStep, in2 := #JOB_4_STEP_01)
      Contact( "Unit1.Em3.ControlNodes".webGuid.sequence.status.seqActive )
      wire#w1
      Coil( "Unit1.Em3.ControlNodes".webGuid."step".action[401] )
   END_RUNG
   RUNG wire#w1
      Coil( "Unit1.Em3.ControlNodes".webGuid."step".transition[401] )
   END_RUNG
   RUNG wire#w1
      Contact( "Unit1.Em3.ControlNodes".webGuid."step".transition[401] )
      { S7_Templates := "time_type := Time" } #statTonTimer[401].TON(pt := #SeqDelayTime, et =>)
      Move(in := #JOB_4_STEP_11, out1 => "Unit1.Em3.ControlNodes".webGuid.sequence.status.nextStep)
   END_RUNG
   // the same network as SCL:
   "Unit1.Em3.ControlNodes".webGuid."step".action[401] := ("Unit1.Em3.ControlNodes".webGuid.sequence.status.currentStep = #JOB_4_STEP_01) AND "Unit1.Em3.ControlNodes".webGuid.sequence.status.seqActive;
   "Unit1.Em3.ControlNodes".webGuid."step".transition[401] := ("Unit1.Em3.ControlNodes".webGuid.sequence.status.currentStep = #JOB_4_STEP_01) AND "Unit1.Em3.ControlNodes".webGuid.sequence.status.seqActive;
   #statTonTimer[401].TON(IN := ("Unit1.Em3.ControlNodes".webGuid.sequence.status.currentStep = #JOB_4_STEP_01) AND "Unit1.Em3.ControlNodes".webGuid.sequence.status.seqActive AND "Unit1.Em3.ControlNodes".webGuid."step".transition[401],
                          PT := #SeqDelayTime);
   IF #statTonTimer[401].Q THEN
       "Unit1.Em3.ControlNodes".webGuid.sequence.status.nextStep := #JOB_4_STEP_11;
   END_IF;
END_REGION

REGION Network 29: Step [411] : ReelCutMain Stop Command
   RUNG wire#powerrail
      { S7_Templates := "SrcType := DInt" } EQ_Contact(in1 := "Unit1.Em3.ControlNodes".webGuid.sequence.status.currentStep, in2 := #JOB_4_STEP_11)
      Contact( "Unit1.Em3.ControlNodes".webGuid.sequence.status.seqActive )
      wire#w1
      Coil( "Unit1.Em3.ControlNodes".webGuid."step".action[411] )
   END_RUNG
   RUNG wire#w1
      Contact( "Unit1.MotionNodes".PLCToMotion.Commands.ReelCutMain.CycleStop )
      Contact( "Unit1.MotionNodes".MotionToPLC.Stauts.ReelCutMain.Done )
      Coil( "Unit1.Em3.ControlNodes".webGuid."step".transition[411] )
   END_RUNG
   RUNG wire#w1
      Contact( "Unit1.Em3.ControlNodes".webGuid."step".transition[411] )
      { S7_Templates := "time_type := Time" } #statTonTimer[411].TON(pt := #SeqDelayTime, et =>)
      Move(in := #JOB_4_STEP_21, out1 => "Unit1.Em3.ControlNodes".webGuid.sequence.status.nextStep)
   END_RUNG
   // the same network as SCL:
   "Unit1.Em3.ControlNodes".webGuid."step".action[411] := ("Unit1.Em3.ControlNodes".webGuid.sequence.status.currentStep = #JOB_4_STEP_11) AND "Unit1.Em3.ControlNodes".webGuid.sequence.status.seqActive;
   "Unit1.Em3.ControlNodes".webGuid."step".transition[411] := ("Unit1.Em3.ControlNodes".webGuid.sequence.status.currentStep = #JOB_4_STEP_11) AND "Unit1.Em3.ControlNodes".webGuid.sequence.status.seqActive AND "Unit1.MotionNodes".PLCToMotion.Commands.ReelCutMain.CycleStop AND "Unit1.MotionNodes".MotionToPLC.Stauts.ReelCutMain.Done;
   #statTonTimer[411].TON(IN := ("Unit1.Em3.ControlNodes".webGuid.sequence.status.currentStep = #JOB_4_STEP_11) AND "Unit1.Em3.ControlNodes".webGuid.sequence.status.seqActive AND "Unit1.Em3.ControlNodes".webGuid."step".transition[411],
                          PT := #SeqDelayTime);
   IF #statTonTimer[411].Q THEN
       "Unit1.Em3.ControlNodes".webGuid.sequence.status.nextStep := #JOB_4_STEP_21;
   END_IF;
END_REGION

REGION Network 30: Step [421] : ReelCutMain Done Delay
   RUNG wire#powerrail
      { S7_Templates := "SrcType := DInt" } EQ_Contact(in1 := "Unit1.Em3.ControlNodes".webGuid.sequence.status.currentStep, in2 := #JOB_4_STEP_21)
      Contact( "Unit1.Em3.ControlNodes".webGuid.sequence.status.seqActive )
      wire#w1
      Coil( "Unit1.Em3.ControlNodes".webGuid."step".action[421] )
   END_RUNG
   RUNG wire#w1
      I_Contact( "Unit1.MotionNodes".MotionToPLC.Stauts.ReelCutMain.Done )
      Coil( "Unit1.Em3.ControlNodes".webGuid."step".transition[421] )
   END_RUNG
   RUNG wire#w1
      Contact( "Unit1.Em3.ControlNodes".webGuid."step".transition[421] )
      { S7_Templates := "time_type := Time" } #statTonTimer[421].TON(pt := #SeqDelayTime, et =>)
      Move(in := #JOB_4_STEP_31, out1 => "Unit1.Em3.ControlNodes".webGuid.sequence.status.nextStep)
   END_RUNG
   // the same network as SCL:
   "Unit1.Em3.ControlNodes".webGuid."step".action[421] := ("Unit1.Em3.ControlNodes".webGuid.sequence.status.currentStep = #JOB_4_STEP_21) AND "Unit1.Em3.ControlNodes".webGuid.sequence.status.seqActive;
   "Unit1.Em3.ControlNodes".webGuid."step".transition[421] := ("Unit1.Em3.ControlNodes".webGuid.sequence.status.currentStep = #JOB_4_STEP_21) AND "Unit1.Em3.ControlNodes".webGuid.sequence.status.seqActive AND NOT "Unit1.MotionNodes".MotionToPLC.Stauts.ReelCutMain.Done;
   #statTonTimer[421].TON(IN := ("Unit1.Em3.ControlNodes".webGuid.sequence.status.currentStep = #JOB_4_STEP_21) AND "Unit1.Em3.ControlNodes".webGuid.sequence.status.seqActive AND "Unit1.Em3.ControlNodes".webGuid."step".transition[421],
                          PT := #SeqDelayTime);
   IF #statTonTimer[421].Q THEN
       "Unit1.Em3.ControlNodes".webGuid.sequence.status.nextStep := #JOB_4_STEP_31;
   END_IF;
END_REGION

REGION Network 31: Step [431] : ReelCutMain FullStep Command
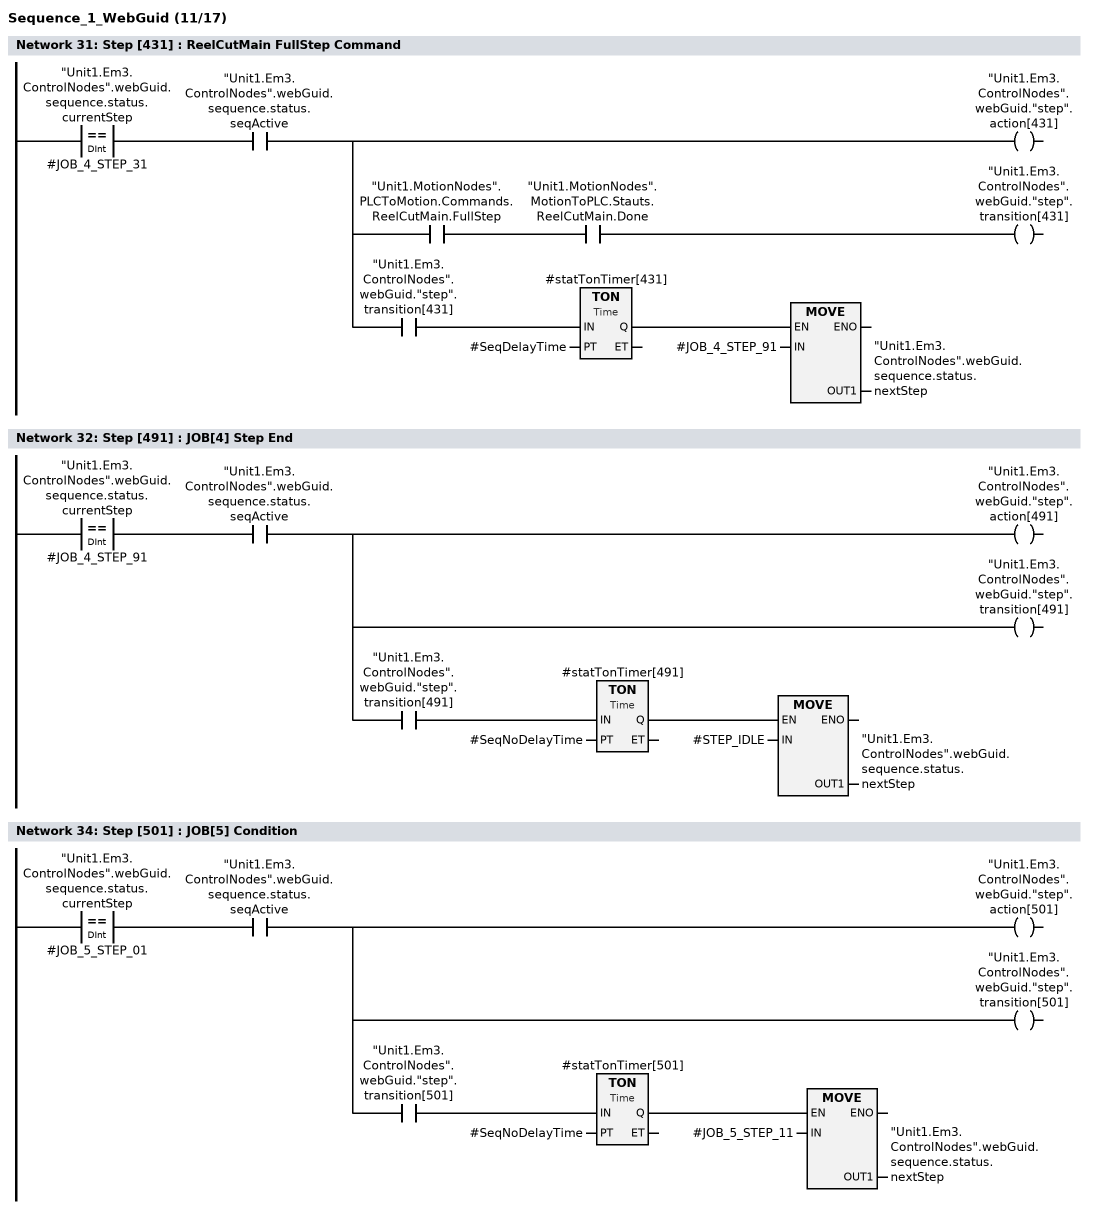
   RUNG wire#powerrail
      { S7_Templates := "SrcType := DInt" } EQ_Contact(in1 := "Unit1.Em3.ControlNodes".webGuid.sequence.status.currentStep, in2 := #JOB_4_STEP_31)
      Contact( "Unit1.Em3.ControlNodes".webGuid.sequence.status.seqActive )
      wire#w1
      Coil( "Unit1.Em3.ControlNodes".webGuid."step".action[431] )
   END_RUNG
   RUNG wire#w1
      Contact( "Unit1.MotionNodes".PLCToMotion.Commands.ReelCutMain.FullStep )
      Contact( "Unit1.MotionNodes".MotionToPLC.Stauts.ReelCutMain.Done )
      Coil( "Unit1.Em3.ControlNodes".webGuid."step".transition[431] )
   END_RUNG
   RUNG wire#w1
      Contact( "Unit1.Em3.ControlNodes".webGuid."step".transition[431] )
      { S7_Templates := "time_type := Time" } #statTonTimer[431].TON(pt := #SeqDelayTime, et =>)
      Move(in := #JOB_4_STEP_91, out1 => "Unit1.Em3.ControlNodes".webGuid.sequence.status.nextStep)
   END_RUNG
   // the same network as SCL:
   "Unit1.Em3.ControlNodes".webGuid."step".action[431] := ("Unit1.Em3.ControlNodes".webGuid.sequence.status.currentStep = #JOB_4_STEP_31) AND "Unit1.Em3.ControlNodes".webGuid.sequence.status.seqActive;
   "Unit1.Em3.ControlNodes".webGuid."step".transition[431] := ("Unit1.Em3.ControlNodes".webGuid.sequence.status.currentStep = #JOB_4_STEP_31) AND "Unit1.Em3.ControlNodes".webGuid.sequence.status.seqActive AND "Unit1.MotionNodes".PLCToMotion.Commands.ReelCutMain.FullStep AND "Unit1.MotionNodes".MotionToPLC.Stauts.ReelCutMain.Done;
   #statTonTimer[431].TON(IN := ("Unit1.Em3.ControlNodes".webGuid.sequence.status.currentStep = #JOB_4_STEP_31) AND "Unit1.Em3.ControlNodes".webGuid.sequence.status.seqActive AND "Unit1.Em3.ControlNodes".webGuid."step".transition[431],
                          PT := #SeqDelayTime);
   IF #statTonTimer[431].Q THEN
       "Unit1.Em3.ControlNodes".webGuid.sequence.status.nextStep := #JOB_4_STEP_91;
   END_IF;
END_REGION

REGION Network 32: Step [491] : JOB[4] Step End
   RUNG wire#powerrail
      { S7_Templates := "SrcType := DInt" } EQ_Contact(in1 := "Unit1.Em3.ControlNodes".webGuid.sequence.status.currentStep, in2 := #JOB_4_STEP_91)
      Contact( "Unit1.Em3.ControlNodes".webGuid.sequence.status.seqActive )
      wire#w1
      Coil( "Unit1.Em3.ControlNodes".webGuid."step".action[491] )
   END_RUNG
   RUNG wire#w1
      Coil( "Unit1.Em3.ControlNodes".webGuid."step".transition[491] )
   END_RUNG
   RUNG wire#w1
      Contact( "Unit1.Em3.ControlNodes".webGuid."step".transition[491] )
      { S7_Templates := "time_type := Time" } #statTonTimer[491].TON(pt := #SeqNoDelayTime, et =>)
      Move(in := #STEP_IDLE, out1 => "Unit1.Em3.ControlNodes".webGuid.sequence.status.nextStep)
   END_RUNG
   // the same network as SCL:
   "Unit1.Em3.ControlNodes".webGuid."step".action[491] := ("Unit1.Em3.ControlNodes".webGuid.sequence.status.currentStep = #JOB_4_STEP_91) AND "Unit1.Em3.ControlNodes".webGuid.sequence.status.seqActive;
   "Unit1.Em3.ControlNodes".webGuid."step".transition[491] := ("Unit1.Em3.ControlNodes".webGuid.sequence.status.currentStep = #JOB_4_STEP_91) AND "Unit1.Em3.ControlNodes".webGuid.sequence.status.seqActive;
   #statTonTimer[491].TON(IN := ("Unit1.Em3.ControlNodes".webGuid.sequence.status.currentStep = #JOB_4_STEP_91) AND "Unit1.Em3.ControlNodes".webGuid.sequence.status.seqActive AND "Unit1.Em3.ControlNodes".webGuid."step".transition[491],
                          PT := #SeqNoDelayTime);
   IF #statTonTimer[491].Q THEN
       "Unit1.Em3.ControlNodes".webGuid.sequence.status.nextStep := #STEP_IDLE;
   END_IF;
END_REGION

REGION Network 33: ******************** JOB[5] MOTION AUTO ********************
END_REGION

REGION Network 34: Step [501] : JOB[5] Condition
   RUNG wire#powerrail
      { S7_Templates := "SrcType := DInt" } EQ_Contact(in1 := "Unit1.Em3.ControlNodes".webGuid.sequence.status.currentStep, in2 := #JOB_5_STEP_01)
      Contact( "Unit1.Em3.ControlNodes".webGuid.sequence.status.seqActive )
      wire#w1
      Coil( "Unit1.Em3.ControlNodes".webGuid."step".action[501] )
   END_RUNG
   RUNG wire#w1
      Coil( "Unit1.Em3.ControlNodes".webGuid."step".transition[501] )
   END_RUNG
   RUNG wire#w1
      Contact( "Unit1.Em3.ControlNodes".webGuid."step".transition[501] )
      { S7_Templates := "time_type := Time" } #statTonTimer[501].TON(pt := #SeqNoDelayTime, et =>)
      Move(in := #JOB_5_STEP_11, out1 => "Unit1.Em3.ControlNodes".webGuid.sequence.status.nextStep)
   END_RUNG
   // the same network as SCL:
   "Unit1.Em3.ControlNodes".webGuid."step".action[501] := ("Unit1.Em3.ControlNodes".webGuid.sequence.status.currentStep = #JOB_5_STEP_01) AND "Unit1.Em3.ControlNodes".webGuid.sequence.status.seqActive;
   "Unit1.Em3.ControlNodes".webGuid."step".transition[501] := ("Unit1.Em3.ControlNodes".webGuid.sequence.status.currentStep = #JOB_5_STEP_01) AND "Unit1.Em3.ControlNodes".webGuid.sequence.status.seqActive;
   #statTonTimer[501].TON(IN := ("Unit1.Em3.ControlNodes".webGuid.sequence.status.currentStep = #JOB_5_STEP_01) AND "Unit1.Em3.ControlNodes".webGuid.sequence.status.seqActive AND "Unit1.Em3.ControlNodes".webGuid."step".transition[501],
                          PT := #SeqNoDelayTime);
   IF #statTonTimer[501].Q THEN
       "Unit1.Em3.ControlNodes".webGuid.sequence.status.nextStep := #JOB_5_STEP_11;
   END_IF;
END_REGION

REGION Network 35: Step [511] : ReelCutMain Stop Command
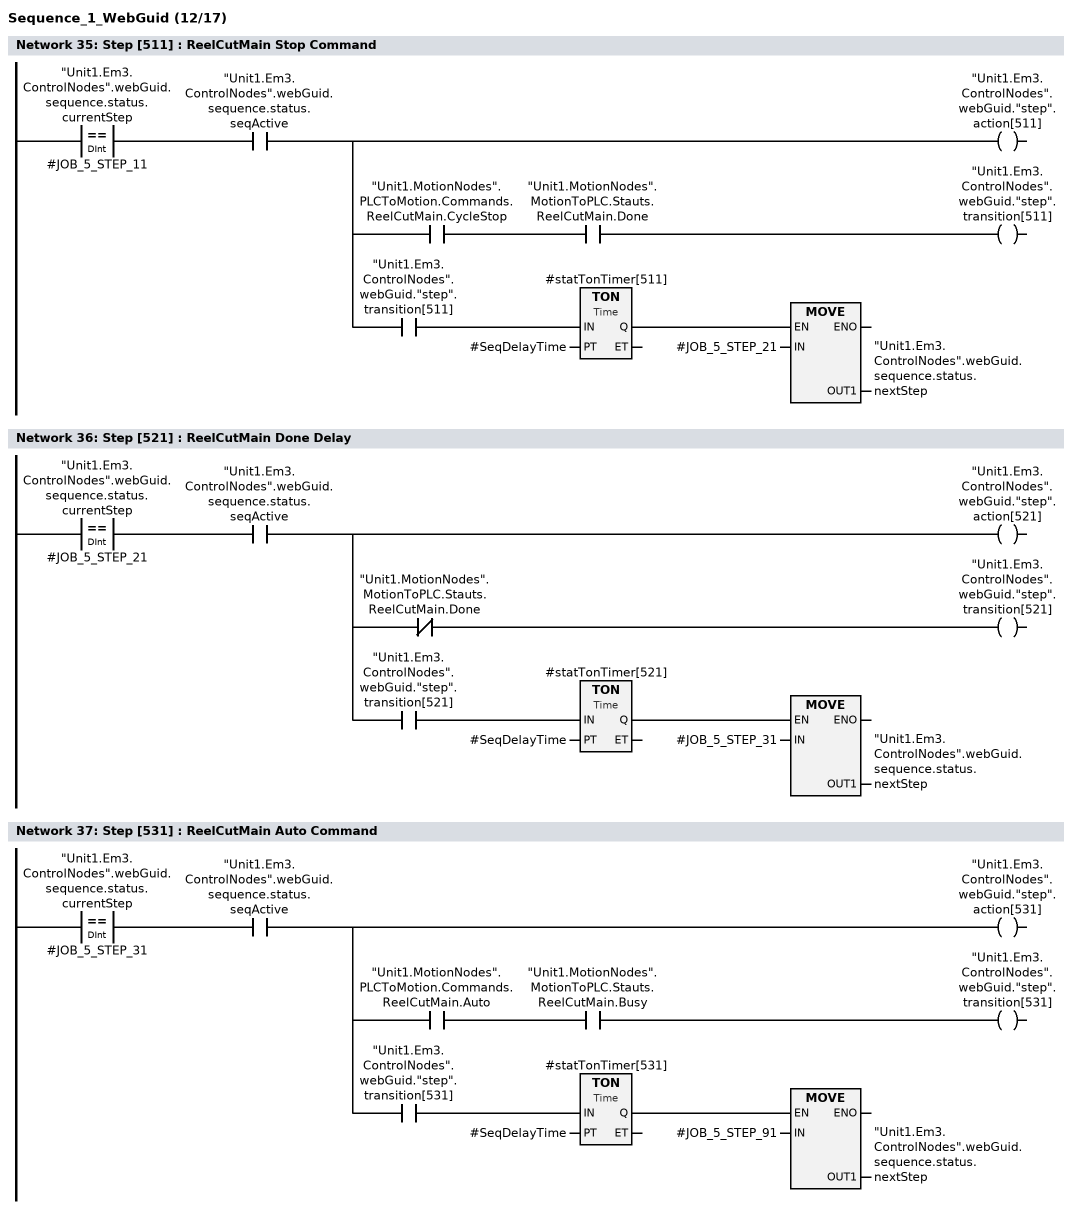
   RUNG wire#powerrail
      { S7_Templates := "SrcType := DInt" } EQ_Contact(in1 := "Unit1.Em3.ControlNodes".webGuid.sequence.status.currentStep, in2 := #JOB_5_STEP_11)
      Contact( "Unit1.Em3.ControlNodes".webGuid.sequence.status.seqActive )
      wire#w1
      Coil( "Unit1.Em3.ControlNodes".webGuid."step".action[511] )
   END_RUNG
   RUNG wire#w1
      Contact( "Unit1.MotionNodes".PLCToMotion.Commands.ReelCutMain.CycleStop )
      Contact( "Unit1.MotionNodes".MotionToPLC.Stauts.ReelCutMain.Done )
      Coil( "Unit1.Em3.ControlNodes".webGuid."step".transition[511] )
   END_RUNG
   RUNG wire#w1
      Contact( "Unit1.Em3.ControlNodes".webGuid."step".transition[511] )
      { S7_Templates := "time_type := Time" } #statTonTimer[511].TON(pt := #SeqDelayTime, et =>)
      Move(in := #JOB_5_STEP_21, out1 => "Unit1.Em3.ControlNodes".webGuid.sequence.status.nextStep)
   END_RUNG
   // the same network as SCL:
   "Unit1.Em3.ControlNodes".webGuid."step".action[511] := ("Unit1.Em3.ControlNodes".webGuid.sequence.status.currentStep = #JOB_5_STEP_11) AND "Unit1.Em3.ControlNodes".webGuid.sequence.status.seqActive;
   "Unit1.Em3.ControlNodes".webGuid."step".transition[511] := ("Unit1.Em3.ControlNodes".webGuid.sequence.status.currentStep = #JOB_5_STEP_11) AND "Unit1.Em3.ControlNodes".webGuid.sequence.status.seqActive AND "Unit1.MotionNodes".PLCToMotion.Commands.ReelCutMain.CycleStop AND "Unit1.MotionNodes".MotionToPLC.Stauts.ReelCutMain.Done;
   #statTonTimer[511].TON(IN := ("Unit1.Em3.ControlNodes".webGuid.sequence.status.currentStep = #JOB_5_STEP_11) AND "Unit1.Em3.ControlNodes".webGuid.sequence.status.seqActive AND "Unit1.Em3.ControlNodes".webGuid."step".transition[511],
                          PT := #SeqDelayTime);
   IF #statTonTimer[511].Q THEN
       "Unit1.Em3.ControlNodes".webGuid.sequence.status.nextStep := #JOB_5_STEP_21;
   END_IF;
END_REGION

REGION Network 36: Step [521] : ReelCutMain Done Delay
   RUNG wire#powerrail
      { S7_Templates := "SrcType := DInt" } EQ_Contact(in1 := "Unit1.Em3.ControlNodes".webGuid.sequence.status.currentStep, in2 := #JOB_5_STEP_21)
      Contact( "Unit1.Em3.ControlNodes".webGuid.sequence.status.seqActive )
      wire#w1
      Coil( "Unit1.Em3.ControlNodes".webGuid."step".action[521] )
   END_RUNG
   RUNG wire#w1
      I_Contact( "Unit1.MotionNodes".MotionToPLC.Stauts.ReelCutMain.Done )
      Coil( "Unit1.Em3.ControlNodes".webGuid."step".transition[521] )
   END_RUNG
   RUNG wire#w1
      Contact( "Unit1.Em3.ControlNodes".webGuid."step".transition[521] )
      { S7_Templates := "time_type := Time" } #statTonTimer[521].TON(pt := #SeqDelayTime, et =>)
      Move(in := #JOB_5_STEP_31, out1 => "Unit1.Em3.ControlNodes".webGuid.sequence.status.nextStep)
   END_RUNG
   // the same network as SCL:
   "Unit1.Em3.ControlNodes".webGuid."step".action[521] := ("Unit1.Em3.ControlNodes".webGuid.sequence.status.currentStep = #JOB_5_STEP_21) AND "Unit1.Em3.ControlNodes".webGuid.sequence.status.seqActive;
   "Unit1.Em3.ControlNodes".webGuid."step".transition[521] := ("Unit1.Em3.ControlNodes".webGuid.sequence.status.currentStep = #JOB_5_STEP_21) AND "Unit1.Em3.ControlNodes".webGuid.sequence.status.seqActive AND NOT "Unit1.MotionNodes".MotionToPLC.Stauts.ReelCutMain.Done;
   #statTonTimer[521].TON(IN := ("Unit1.Em3.ControlNodes".webGuid.sequence.status.currentStep = #JOB_5_STEP_21) AND "Unit1.Em3.ControlNodes".webGuid.sequence.status.seqActive AND "Unit1.Em3.ControlNodes".webGuid."step".transition[521],
                          PT := #SeqDelayTime);
   IF #statTonTimer[521].Q THEN
       "Unit1.Em3.ControlNodes".webGuid.sequence.status.nextStep := #JOB_5_STEP_31;
   END_IF;
END_REGION

REGION Network 37: Step [531] : ReelCutMain Auto Command
   RUNG wire#powerrail
      { S7_Templates := "SrcType := DInt" } EQ_Contact(in1 := "Unit1.Em3.ControlNodes".webGuid.sequence.status.currentStep, in2 := #JOB_5_STEP_31)
      Contact( "Unit1.Em3.ControlNodes".webGuid.sequence.status.seqActive )
      wire#w1
      Coil( "Unit1.Em3.ControlNodes".webGuid."step".action[531] )
   END_RUNG
   RUNG wire#w1
      Contact( "Unit1.MotionNodes".PLCToMotion.Commands.ReelCutMain.Auto )
      Contact( "Unit1.MotionNodes".MotionToPLC.Stauts.ReelCutMain.Busy )
      Coil( "Unit1.Em3.ControlNodes".webGuid."step".transition[531] )
   END_RUNG
   RUNG wire#w1
      Contact( "Unit1.Em3.ControlNodes".webGuid."step".transition[531] )
      { S7_Templates := "time_type := Time" } #statTonTimer[531].TON(pt := #SeqDelayTime, et =>)
      Move(in := #JOB_5_STEP_91, out1 => "Unit1.Em3.ControlNodes".webGuid.sequence.status.nextStep)
   END_RUNG
   // the same network as SCL:
   "Unit1.Em3.ControlNodes".webGuid."step".action[531] := ("Unit1.Em3.ControlNodes".webGuid.sequence.status.currentStep = #JOB_5_STEP_31) AND "Unit1.Em3.ControlNodes".webGuid.sequence.status.seqActive;
   "Unit1.Em3.ControlNodes".webGuid."step".transition[531] := ("Unit1.Em3.ControlNodes".webGuid.sequence.status.currentStep = #JOB_5_STEP_31) AND "Unit1.Em3.ControlNodes".webGuid.sequence.status.seqActive AND "Unit1.MotionNodes".PLCToMotion.Commands.ReelCutMain.Auto AND "Unit1.MotionNodes".MotionToPLC.Stauts.ReelCutMain.Busy;
   #statTonTimer[531].TON(IN := ("Unit1.Em3.ControlNodes".webGuid.sequence.status.currentStep = #JOB_5_STEP_31) AND "Unit1.Em3.ControlNodes".webGuid.sequence.status.seqActive AND "Unit1.Em3.ControlNodes".webGuid."step".transition[531],
                          PT := #SeqDelayTime);
   IF #statTonTimer[531].Q THEN
       "Unit1.Em3.ControlNodes".webGuid.sequence.status.nextStep := #JOB_5_STEP_91;
   END_IF;
END_REGION

REGION Network 38: Step [591] : JOB[5] Step End
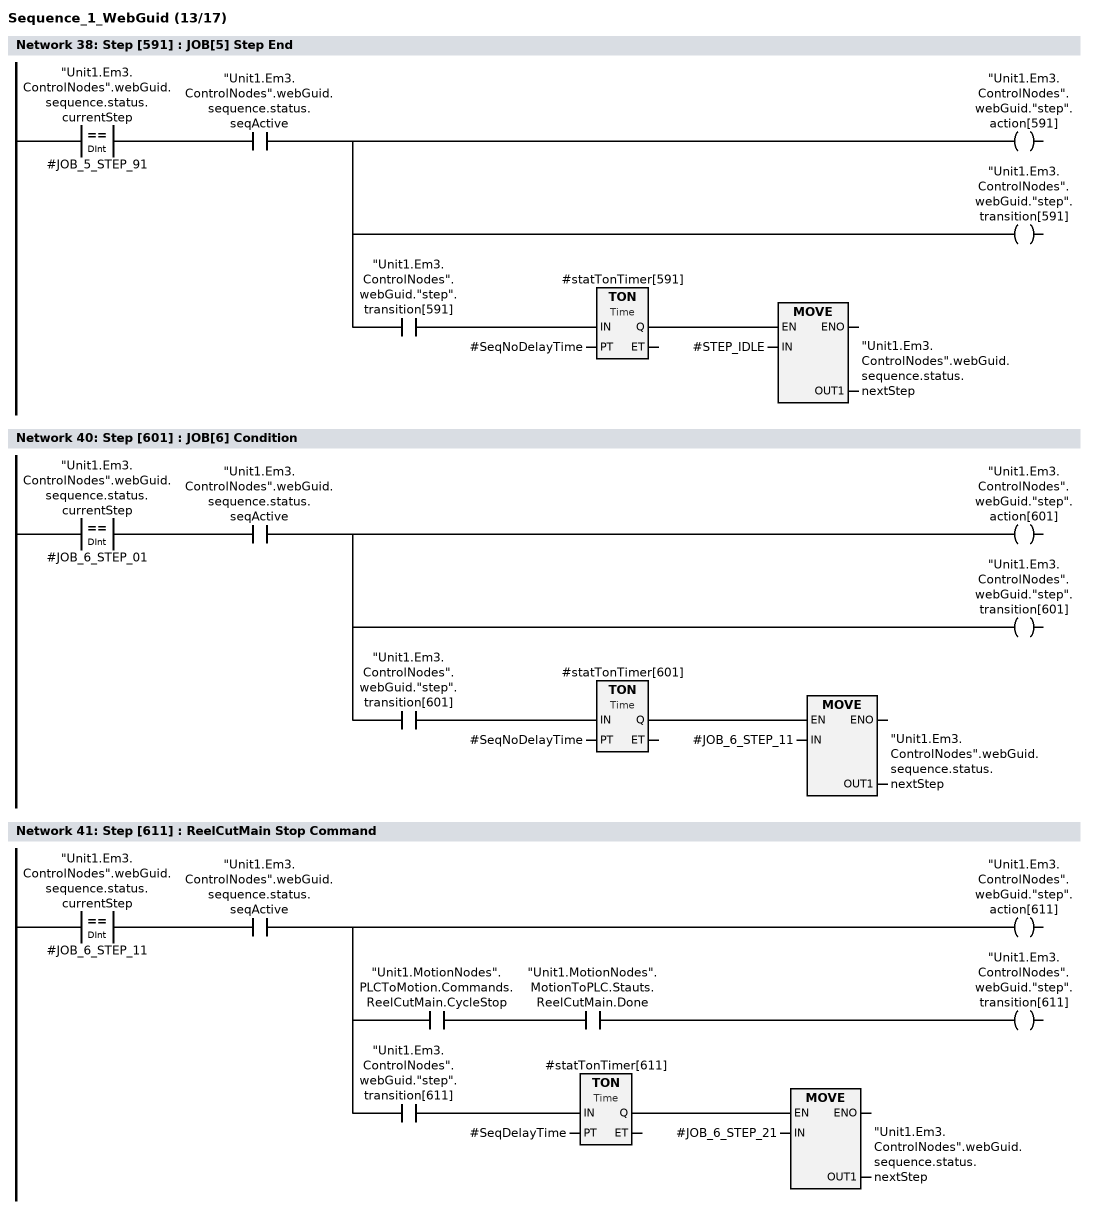
   RUNG wire#powerrail
      { S7_Templates := "SrcType := DInt" } EQ_Contact(in1 := "Unit1.Em3.ControlNodes".webGuid.sequence.status.currentStep, in2 := #JOB_5_STEP_91)
      Contact( "Unit1.Em3.ControlNodes".webGuid.sequence.status.seqActive )
      wire#w1
      Coil( "Unit1.Em3.ControlNodes".webGuid."step".action[591] )
   END_RUNG
   RUNG wire#w1
      Coil( "Unit1.Em3.ControlNodes".webGuid."step".transition[591] )
   END_RUNG
   RUNG wire#w1
      Contact( "Unit1.Em3.ControlNodes".webGuid."step".transition[591] )
      { S7_Templates := "time_type := Time" } #statTonTimer[591].TON(pt := #SeqNoDelayTime, et =>)
      Move(in := #STEP_IDLE, out1 => "Unit1.Em3.ControlNodes".webGuid.sequence.status.nextStep)
   END_RUNG
   // the same network as SCL:
   "Unit1.Em3.ControlNodes".webGuid."step".action[591] := ("Unit1.Em3.ControlNodes".webGuid.sequence.status.currentStep = #JOB_5_STEP_91) AND "Unit1.Em3.ControlNodes".webGuid.sequence.status.seqActive;
   "Unit1.Em3.ControlNodes".webGuid."step".transition[591] := ("Unit1.Em3.ControlNodes".webGuid.sequence.status.currentStep = #JOB_5_STEP_91) AND "Unit1.Em3.ControlNodes".webGuid.sequence.status.seqActive;
   #statTonTimer[591].TON(IN := ("Unit1.Em3.ControlNodes".webGuid.sequence.status.currentStep = #JOB_5_STEP_91) AND "Unit1.Em3.ControlNodes".webGuid.sequence.status.seqActive AND "Unit1.Em3.ControlNodes".webGuid."step".transition[591],
                          PT := #SeqNoDelayTime);
   IF #statTonTimer[591].Q THEN
       "Unit1.Em3.ControlNodes".webGuid.sequence.status.nextStep := #STEP_IDLE;
   END_IF;
END_REGION

REGION Network 39: ******************** JOB[6] MOTION SEMI STEP ********************
END_REGION

REGION Network 40: Step [601] : JOB[6] Condition
   RUNG wire#powerrail
      { S7_Templates := "SrcType := DInt" } EQ_Contact(in1 := "Unit1.Em3.ControlNodes".webGuid.sequence.status.currentStep, in2 := #JOB_6_STEP_01)
      Contact( "Unit1.Em3.ControlNodes".webGuid.sequence.status.seqActive )
      wire#w1
      Coil( "Unit1.Em3.ControlNodes".webGuid."step".action[601] )
   END_RUNG
   RUNG wire#w1
      Coil( "Unit1.Em3.ControlNodes".webGuid."step".transition[601] )
   END_RUNG
   RUNG wire#w1
      Contact( "Unit1.Em3.ControlNodes".webGuid."step".transition[601] )
      { S7_Templates := "time_type := Time" } #statTonTimer[601].TON(pt := #SeqNoDelayTime, et =>)
      Move(in := #JOB_6_STEP_11, out1 => "Unit1.Em3.ControlNodes".webGuid.sequence.status.nextStep)
   END_RUNG
   // the same network as SCL:
   "Unit1.Em3.ControlNodes".webGuid."step".action[601] := ("Unit1.Em3.ControlNodes".webGuid.sequence.status.currentStep = #JOB_6_STEP_01) AND "Unit1.Em3.ControlNodes".webGuid.sequence.status.seqActive;
   "Unit1.Em3.ControlNodes".webGuid."step".transition[601] := ("Unit1.Em3.ControlNodes".webGuid.sequence.status.currentStep = #JOB_6_STEP_01) AND "Unit1.Em3.ControlNodes".webGuid.sequence.status.seqActive;
   #statTonTimer[601].TON(IN := ("Unit1.Em3.ControlNodes".webGuid.sequence.status.currentStep = #JOB_6_STEP_01) AND "Unit1.Em3.ControlNodes".webGuid.sequence.status.seqActive AND "Unit1.Em3.ControlNodes".webGuid."step".transition[601],
                          PT := #SeqNoDelayTime);
   IF #statTonTimer[601].Q THEN
       "Unit1.Em3.ControlNodes".webGuid.sequence.status.nextStep := #JOB_6_STEP_11;
   END_IF;
END_REGION

REGION Network 41: Step [611] : ReelCutMain Stop Command
   RUNG wire#powerrail
      { S7_Templates := "SrcType := DInt" } EQ_Contact(in1 := "Unit1.Em3.ControlNodes".webGuid.sequence.status.currentStep, in2 := #JOB_6_STEP_11)
      Contact( "Unit1.Em3.ControlNodes".webGuid.sequence.status.seqActive )
      wire#w1
      Coil( "Unit1.Em3.ControlNodes".webGuid."step".action[611] )
   END_RUNG
   RUNG wire#w1
      Contact( "Unit1.MotionNodes".PLCToMotion.Commands.ReelCutMain.CycleStop )
      Contact( "Unit1.MotionNodes".MotionToPLC.Stauts.ReelCutMain.Done )
      Coil( "Unit1.Em3.ControlNodes".webGuid."step".transition[611] )
   END_RUNG
   RUNG wire#w1
      Contact( "Unit1.Em3.ControlNodes".webGuid."step".transition[611] )
      { S7_Templates := "time_type := Time" } #statTonTimer[611].TON(pt := #SeqDelayTime, et =>)
      Move(in := #JOB_6_STEP_21, out1 => "Unit1.Em3.ControlNodes".webGuid.sequence.status.nextStep)
   END_RUNG
   // the same network as SCL:
   "Unit1.Em3.ControlNodes".webGuid."step".action[611] := ("Unit1.Em3.ControlNodes".webGuid.sequence.status.currentStep = #JOB_6_STEP_11) AND "Unit1.Em3.ControlNodes".webGuid.sequence.status.seqActive;
   "Unit1.Em3.ControlNodes".webGuid."step".transition[611] := ("Unit1.Em3.ControlNodes".webGuid.sequence.status.currentStep = #JOB_6_STEP_11) AND "Unit1.Em3.ControlNodes".webGuid.sequence.status.seqActive AND "Unit1.MotionNodes".PLCToMotion.Commands.ReelCutMain.CycleStop AND "Unit1.MotionNodes".MotionToPLC.Stauts.ReelCutMain.Done;
   #statTonTimer[611].TON(IN := ("Unit1.Em3.ControlNodes".webGuid.sequence.status.currentStep = #JOB_6_STEP_11) AND "Unit1.Em3.ControlNodes".webGuid.sequence.status.seqActive AND "Unit1.Em3.ControlNodes".webGuid."step".transition[611],
                          PT := #SeqDelayTime);
   IF #statTonTimer[611].Q THEN
       "Unit1.Em3.ControlNodes".webGuid.sequence.status.nextStep := #JOB_6_STEP_21;
   END_IF;
END_REGION

REGION Network 42: Step [621] : ReelCutMain Done Delay
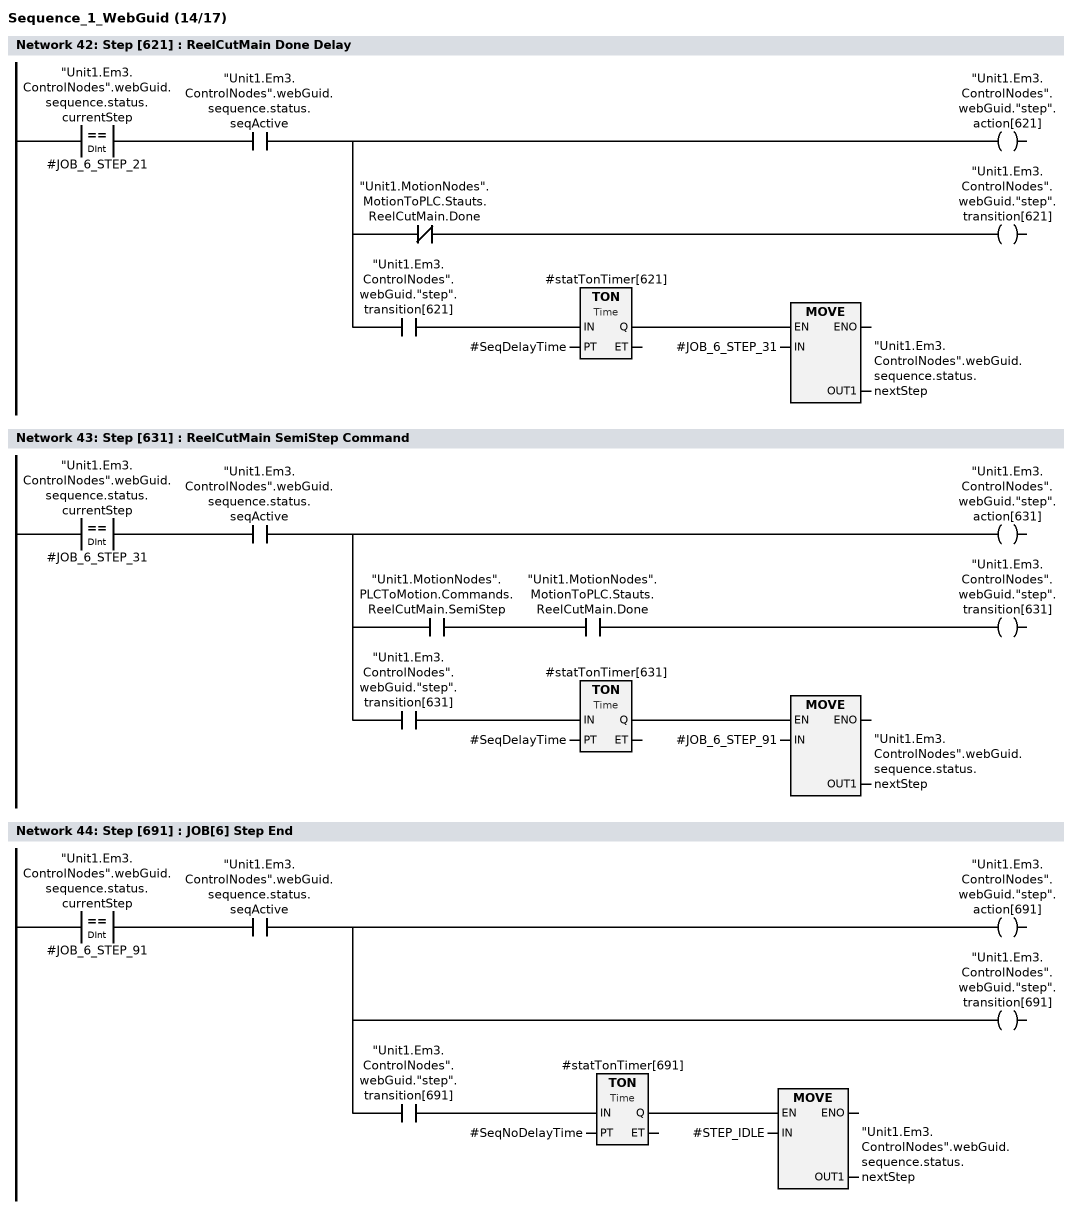
   RUNG wire#powerrail
      { S7_Templates := "SrcType := DInt" } EQ_Contact(in1 := "Unit1.Em3.ControlNodes".webGuid.sequence.status.currentStep, in2 := #JOB_6_STEP_21)
      Contact( "Unit1.Em3.ControlNodes".webGuid.sequence.status.seqActive )
      wire#w1
      Coil( "Unit1.Em3.ControlNodes".webGuid."step".action[621] )
   END_RUNG
   RUNG wire#w1
      I_Contact( "Unit1.MotionNodes".MotionToPLC.Stauts.ReelCutMain.Done )
      Coil( "Unit1.Em3.ControlNodes".webGuid."step".transition[621] )
   END_RUNG
   RUNG wire#w1
      Contact( "Unit1.Em3.ControlNodes".webGuid."step".transition[621] )
      { S7_Templates := "time_type := Time" } #statTonTimer[621].TON(pt := #SeqDelayTime, et =>)
      Move(in := #JOB_6_STEP_31, out1 => "Unit1.Em3.ControlNodes".webGuid.sequence.status.nextStep)
   END_RUNG
   // the same network as SCL:
   "Unit1.Em3.ControlNodes".webGuid."step".action[621] := ("Unit1.Em3.ControlNodes".webGuid.sequence.status.currentStep = #JOB_6_STEP_21) AND "Unit1.Em3.ControlNodes".webGuid.sequence.status.seqActive;
   "Unit1.Em3.ControlNodes".webGuid."step".transition[621] := ("Unit1.Em3.ControlNodes".webGuid.sequence.status.currentStep = #JOB_6_STEP_21) AND "Unit1.Em3.ControlNodes".webGuid.sequence.status.seqActive AND NOT "Unit1.MotionNodes".MotionToPLC.Stauts.ReelCutMain.Done;
   #statTonTimer[621].TON(IN := ("Unit1.Em3.ControlNodes".webGuid.sequence.status.currentStep = #JOB_6_STEP_21) AND "Unit1.Em3.ControlNodes".webGuid.sequence.status.seqActive AND "Unit1.Em3.ControlNodes".webGuid."step".transition[621],
                          PT := #SeqDelayTime);
   IF #statTonTimer[621].Q THEN
       "Unit1.Em3.ControlNodes".webGuid.sequence.status.nextStep := #JOB_6_STEP_31;
   END_IF;
END_REGION

REGION Network 43: Step [631] : ReelCutMain SemiStep Command
   RUNG wire#powerrail
      { S7_Templates := "SrcType := DInt" } EQ_Contact(in1 := "Unit1.Em3.ControlNodes".webGuid.sequence.status.currentStep, in2 := #JOB_6_STEP_31)
      Contact( "Unit1.Em3.ControlNodes".webGuid.sequence.status.seqActive )
      wire#w1
      Coil( "Unit1.Em3.ControlNodes".webGuid."step".action[631] )
   END_RUNG
   RUNG wire#w1
      Contact( "Unit1.MotionNodes".PLCToMotion.Commands.ReelCutMain.SemiStep )
      Contact( "Unit1.MotionNodes".MotionToPLC.Stauts.ReelCutMain.Done )
      Coil( "Unit1.Em3.ControlNodes".webGuid."step".transition[631] )
   END_RUNG
   RUNG wire#w1
      Contact( "Unit1.Em3.ControlNodes".webGuid."step".transition[631] )
      { S7_Templates := "time_type := Time" } #statTonTimer[631].TON(pt := #SeqDelayTime, et =>)
      Move(in := #JOB_6_STEP_91, out1 => "Unit1.Em3.ControlNodes".webGuid.sequence.status.nextStep)
   END_RUNG
   // the same network as SCL:
   "Unit1.Em3.ControlNodes".webGuid."step".action[631] := ("Unit1.Em3.ControlNodes".webGuid.sequence.status.currentStep = #JOB_6_STEP_31) AND "Unit1.Em3.ControlNodes".webGuid.sequence.status.seqActive;
   "Unit1.Em3.ControlNodes".webGuid."step".transition[631] := ("Unit1.Em3.ControlNodes".webGuid.sequence.status.currentStep = #JOB_6_STEP_31) AND "Unit1.Em3.ControlNodes".webGuid.sequence.status.seqActive AND "Unit1.MotionNodes".PLCToMotion.Commands.ReelCutMain.SemiStep AND "Unit1.MotionNodes".MotionToPLC.Stauts.ReelCutMain.Done;
   #statTonTimer[631].TON(IN := ("Unit1.Em3.ControlNodes".webGuid.sequence.status.currentStep = #JOB_6_STEP_31) AND "Unit1.Em3.ControlNodes".webGuid.sequence.status.seqActive AND "Unit1.Em3.ControlNodes".webGuid."step".transition[631],
                          PT := #SeqDelayTime);
   IF #statTonTimer[631].Q THEN
       "Unit1.Em3.ControlNodes".webGuid.sequence.status.nextStep := #JOB_6_STEP_91;
   END_IF;
END_REGION

REGION Network 44: Step [691] : JOB[6] Step End
   RUNG wire#powerrail
      { S7_Templates := "SrcType := DInt" } EQ_Contact(in1 := "Unit1.Em3.ControlNodes".webGuid.sequence.status.currentStep, in2 := #JOB_6_STEP_91)
      Contact( "Unit1.Em3.ControlNodes".webGuid.sequence.status.seqActive )
      wire#w1
      Coil( "Unit1.Em3.ControlNodes".webGuid."step".action[691] )
   END_RUNG
   RUNG wire#w1
      Coil( "Unit1.Em3.ControlNodes".webGuid."step".transition[691] )
   END_RUNG
   RUNG wire#w1
      Contact( "Unit1.Em3.ControlNodes".webGuid."step".transition[691] )
      { S7_Templates := "time_type := Time" } #statTonTimer[691].TON(pt := #SeqNoDelayTime, et =>)
      Move(in := #STEP_IDLE, out1 => "Unit1.Em3.ControlNodes".webGuid.sequence.status.nextStep)
   END_RUNG
   // the same network as SCL:
   "Unit1.Em3.ControlNodes".webGuid."step".action[691] := ("Unit1.Em3.ControlNodes".webGuid.sequence.status.currentStep = #JOB_6_STEP_91) AND "Unit1.Em3.ControlNodes".webGuid.sequence.status.seqActive;
   "Unit1.Em3.ControlNodes".webGuid."step".transition[691] := ("Unit1.Em3.ControlNodes".webGuid.sequence.status.currentStep = #JOB_6_STEP_91) AND "Unit1.Em3.ControlNodes".webGuid.sequence.status.seqActive;
   #statTonTimer[691].TON(IN := ("Unit1.Em3.ControlNodes".webGuid.sequence.status.currentStep = #JOB_6_STEP_91) AND "Unit1.Em3.ControlNodes".webGuid.sequence.status.seqActive AND "Unit1.Em3.ControlNodes".webGuid."step".transition[691],
                          PT := #SeqNoDelayTime);
   IF #statTonTimer[691].Q THEN
       "Unit1.Em3.ControlNodes".webGuid.sequence.status.nextStep := #STEP_IDLE;
   END_IF;
END_REGION

REGION Network 45: ******************** JOB[7] MOTION CYCLE STOP ********************
END_REGION

REGION Network 46: Step [701] : JOB[7] Condition
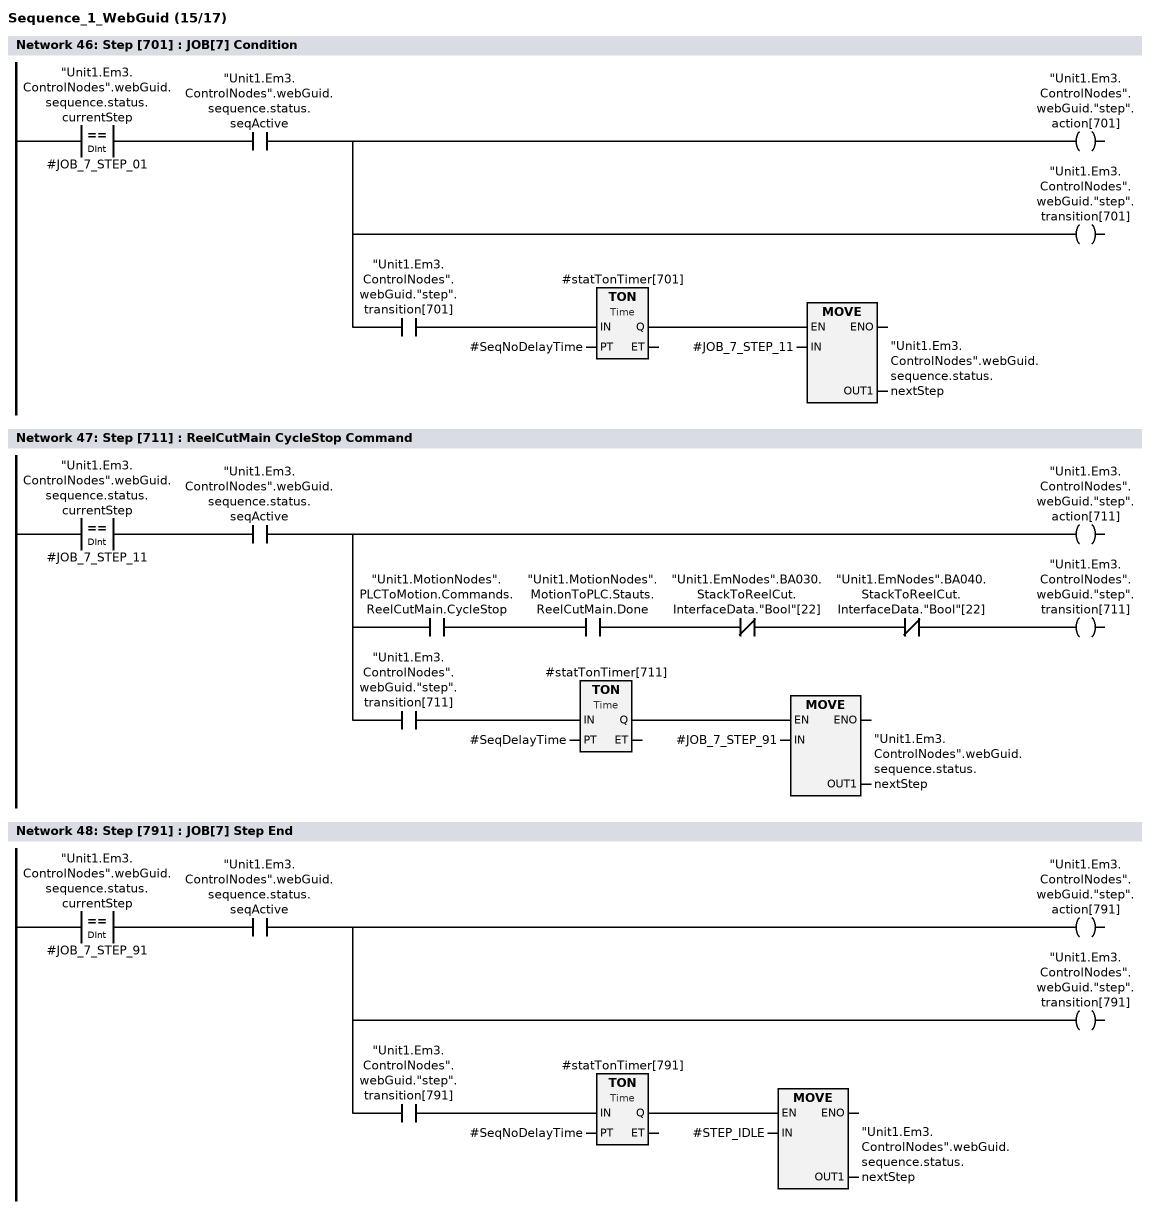
   RUNG wire#powerrail
      { S7_Templates := "SrcType := DInt" } EQ_Contact(in1 := "Unit1.Em3.ControlNodes".webGuid.sequence.status.currentStep, in2 := #JOB_7_STEP_01)
      Contact( "Unit1.Em3.ControlNodes".webGuid.sequence.status.seqActive )
      wire#w1
      Coil( "Unit1.Em3.ControlNodes".webGuid."step".action[701] )
   END_RUNG
   RUNG wire#w1
      Coil( "Unit1.Em3.ControlNodes".webGuid."step".transition[701] )
   END_RUNG
   RUNG wire#w1
      Contact( "Unit1.Em3.ControlNodes".webGuid."step".transition[701] )
      { S7_Templates := "time_type := Time" } #statTonTimer[701].TON(pt := #SeqNoDelayTime, et =>)
      Move(in := #JOB_7_STEP_11, out1 => "Unit1.Em3.ControlNodes".webGuid.sequence.status.nextStep)
   END_RUNG
   // the same network as SCL:
   "Unit1.Em3.ControlNodes".webGuid."step".action[701] := ("Unit1.Em3.ControlNodes".webGuid.sequence.status.currentStep = #JOB_7_STEP_01) AND "Unit1.Em3.ControlNodes".webGuid.sequence.status.seqActive;
   "Unit1.Em3.ControlNodes".webGuid."step".transition[701] := ("Unit1.Em3.ControlNodes".webGuid.sequence.status.currentStep = #JOB_7_STEP_01) AND "Unit1.Em3.ControlNodes".webGuid.sequence.status.seqActive;
   #statTonTimer[701].TON(IN := ("Unit1.Em3.ControlNodes".webGuid.sequence.status.currentStep = #JOB_7_STEP_01) AND "Unit1.Em3.ControlNodes".webGuid.sequence.status.seqActive AND "Unit1.Em3.ControlNodes".webGuid."step".transition[701],
                          PT := #SeqNoDelayTime);
   IF #statTonTimer[701].Q THEN
       "Unit1.Em3.ControlNodes".webGuid.sequence.status.nextStep := #JOB_7_STEP_11;
   END_IF;
END_REGION

REGION Network 47: Step [711] : ReelCutMain CycleStop Command
   RUNG wire#powerrail
      { S7_Templates := "SrcType := DInt" } EQ_Contact(in1 := "Unit1.Em3.ControlNodes".webGuid.sequence.status.currentStep, in2 := #JOB_7_STEP_11)
      Contact( "Unit1.Em3.ControlNodes".webGuid.sequence.status.seqActive )
      wire#w1
      Coil( "Unit1.Em3.ControlNodes".webGuid."step".action[711] )
   END_RUNG
   RUNG wire#w1
      Contact( "Unit1.MotionNodes".PLCToMotion.Commands.ReelCutMain.CycleStop )
      Contact( "Unit1.MotionNodes".MotionToPLC.Stauts.ReelCutMain.Done )
      I_Contact( "Unit1.EmNodes".BA030.StackToReelCut.InterfaceData."Bool"[22] )
      I_Contact( "Unit1.EmNodes".BA040.StackToReelCut.InterfaceData."Bool"[22] )
      Coil( "Unit1.Em3.ControlNodes".webGuid."step".transition[711] )
   END_RUNG
   RUNG wire#w1
      Contact( "Unit1.Em3.ControlNodes".webGuid."step".transition[711] )
      { S7_Templates := "time_type := Time" } #statTonTimer[711].TON(pt := #SeqDelayTime, et =>)
      Move(in := #JOB_7_STEP_91, out1 => "Unit1.Em3.ControlNodes".webGuid.sequence.status.nextStep)
   END_RUNG
   // the same network as SCL:
   "Unit1.Em3.ControlNodes".webGuid."step".action[711] := ("Unit1.Em3.ControlNodes".webGuid.sequence.status.currentStep = #JOB_7_STEP_11) AND "Unit1.Em3.ControlNodes".webGuid.sequence.status.seqActive;
   "Unit1.Em3.ControlNodes".webGuid."step".transition[711] := ("Unit1.Em3.ControlNodes".webGuid.sequence.status.currentStep = #JOB_7_STEP_11) AND "Unit1.Em3.ControlNodes".webGuid.sequence.status.seqActive AND "Unit1.MotionNodes".PLCToMotion.Commands.ReelCutMain.CycleStop AND "Unit1.MotionNodes".MotionToPLC.Stauts.ReelCutMain.Done AND NOT "Unit1.EmNodes".BA030.StackToReelCut.InterfaceData."Bool"[22] AND NOT "Unit1.EmNodes".BA040.StackToReelCut.InterfaceData."Bool"[22];
   #statTonTimer[711].TON(IN := ("Unit1.Em3.ControlNodes".webGuid.sequence.status.currentStep = #JOB_7_STEP_11) AND "Unit1.Em3.ControlNodes".webGuid.sequence.status.seqActive AND "Unit1.Em3.ControlNodes".webGuid."step".transition[711],
                          PT := #SeqDelayTime);
   IF #statTonTimer[711].Q THEN
       "Unit1.Em3.ControlNodes".webGuid.sequence.status.nextStep := #JOB_7_STEP_91;
   END_IF;
END_REGION

REGION Network 48: Step [791] : JOB[7] Step End
   RUNG wire#powerrail
      { S7_Templates := "SrcType := DInt" } EQ_Contact(in1 := "Unit1.Em3.ControlNodes".webGuid.sequence.status.currentStep, in2 := #JOB_7_STEP_91)
      Contact( "Unit1.Em3.ControlNodes".webGuid.sequence.status.seqActive )
      wire#w1
      Coil( "Unit1.Em3.ControlNodes".webGuid."step".action[791] )
   END_RUNG
   RUNG wire#w1
      Coil( "Unit1.Em3.ControlNodes".webGuid."step".transition[791] )
   END_RUNG
   RUNG wire#w1
      Contact( "Unit1.Em3.ControlNodes".webGuid."step".transition[791] )
      { S7_Templates := "time_type := Time" } #statTonTimer[791].TON(pt := #SeqNoDelayTime, et =>)
      Move(in := #STEP_IDLE, out1 => "Unit1.Em3.ControlNodes".webGuid.sequence.status.nextStep)
   END_RUNG
   // the same network as SCL:
   "Unit1.Em3.ControlNodes".webGuid."step".action[791] := ("Unit1.Em3.ControlNodes".webGuid.sequence.status.currentStep = #JOB_7_STEP_91) AND "Unit1.Em3.ControlNodes".webGuid.sequence.status.seqActive;
   "Unit1.Em3.ControlNodes".webGuid."step".transition[791] := ("Unit1.Em3.ControlNodes".webGuid.sequence.status.currentStep = #JOB_7_STEP_91) AND "Unit1.Em3.ControlNodes".webGuid.sequence.status.seqActive;
   #statTonTimer[791].TON(IN := ("Unit1.Em3.ControlNodes".webGuid.sequence.status.currentStep = #JOB_7_STEP_91) AND "Unit1.Em3.ControlNodes".webGuid.sequence.status.seqActive AND "Unit1.Em3.ControlNodes".webGuid."step".transition[791],
                          PT := #SeqNoDelayTime);
   IF #statTonTimer[791].Q THEN
       "Unit1.Em3.ControlNodes".webGuid.sequence.status.nextStep := #STEP_IDLE;
   END_IF;
END_REGION

REGION Network 49: ******************** JOB[8] MOTION FAST STOP ********************
END_REGION

REGION Network 50: Step [801] : JOB[8] Condition
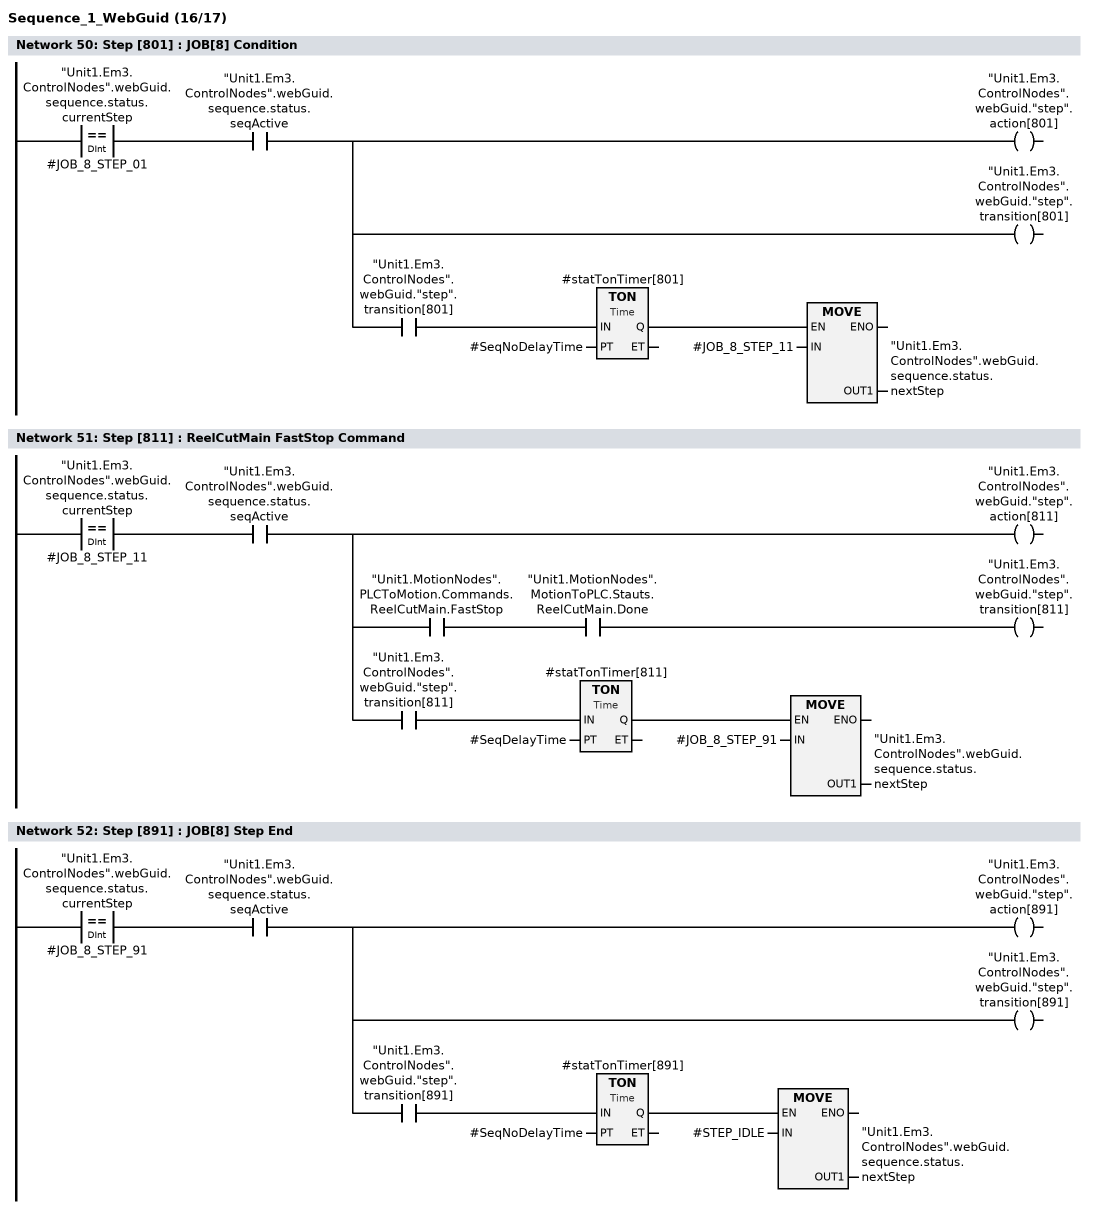
   RUNG wire#powerrail
      { S7_Templates := "SrcType := DInt" } EQ_Contact(in1 := "Unit1.Em3.ControlNodes".webGuid.sequence.status.currentStep, in2 := #JOB_8_STEP_01)
      Contact( "Unit1.Em3.ControlNodes".webGuid.sequence.status.seqActive )
      wire#w1
      Coil( "Unit1.Em3.ControlNodes".webGuid."step".action[801] )
   END_RUNG
   RUNG wire#w1
      Coil( "Unit1.Em3.ControlNodes".webGuid."step".transition[801] )
   END_RUNG
   RUNG wire#w1
      Contact( "Unit1.Em3.ControlNodes".webGuid."step".transition[801] )
      { S7_Templates := "time_type := Time" } #statTonTimer[801].TON(pt := #SeqNoDelayTime, et =>)
      Move(in := #JOB_8_STEP_11, out1 => "Unit1.Em3.ControlNodes".webGuid.sequence.status.nextStep)
   END_RUNG
   // the same network as SCL:
   "Unit1.Em3.ControlNodes".webGuid."step".action[801] := ("Unit1.Em3.ControlNodes".webGuid.sequence.status.currentStep = #JOB_8_STEP_01) AND "Unit1.Em3.ControlNodes".webGuid.sequence.status.seqActive;
   "Unit1.Em3.ControlNodes".webGuid."step".transition[801] := ("Unit1.Em3.ControlNodes".webGuid.sequence.status.currentStep = #JOB_8_STEP_01) AND "Unit1.Em3.ControlNodes".webGuid.sequence.status.seqActive;
   #statTonTimer[801].TON(IN := ("Unit1.Em3.ControlNodes".webGuid.sequence.status.currentStep = #JOB_8_STEP_01) AND "Unit1.Em3.ControlNodes".webGuid.sequence.status.seqActive AND "Unit1.Em3.ControlNodes".webGuid."step".transition[801],
                          PT := #SeqNoDelayTime);
   IF #statTonTimer[801].Q THEN
       "Unit1.Em3.ControlNodes".webGuid.sequence.status.nextStep := #JOB_8_STEP_11;
   END_IF;
END_REGION

REGION Network 51: Step [811] : ReelCutMain FastStop Command
   RUNG wire#powerrail
      { S7_Templates := "SrcType := DInt" } EQ_Contact(in1 := "Unit1.Em3.ControlNodes".webGuid.sequence.status.currentStep, in2 := #JOB_8_STEP_11)
      Contact( "Unit1.Em3.ControlNodes".webGuid.sequence.status.seqActive )
      wire#w1
      Coil( "Unit1.Em3.ControlNodes".webGuid."step".action[811] )
   END_RUNG
   RUNG wire#w1
      Contact( "Unit1.MotionNodes".PLCToMotion.Commands.ReelCutMain.FastStop )
      Contact( "Unit1.MotionNodes".MotionToPLC.Stauts.ReelCutMain.Done )
      Coil( "Unit1.Em3.ControlNodes".webGuid."step".transition[811] )
   END_RUNG
   RUNG wire#w1
      Contact( "Unit1.Em3.ControlNodes".webGuid."step".transition[811] )
      { S7_Templates := "time_type := Time" } #statTonTimer[811].TON(pt := #SeqDelayTime, et =>)
      Move(in := #JOB_8_STEP_91, out1 => "Unit1.Em3.ControlNodes".webGuid.sequence.status.nextStep)
   END_RUNG
   // the same network as SCL:
   "Unit1.Em3.ControlNodes".webGuid."step".action[811] := ("Unit1.Em3.ControlNodes".webGuid.sequence.status.currentStep = #JOB_8_STEP_11) AND "Unit1.Em3.ControlNodes".webGuid.sequence.status.seqActive;
   "Unit1.Em3.ControlNodes".webGuid."step".transition[811] := ("Unit1.Em3.ControlNodes".webGuid.sequence.status.currentStep = #JOB_8_STEP_11) AND "Unit1.Em3.ControlNodes".webGuid.sequence.status.seqActive AND "Unit1.MotionNodes".PLCToMotion.Commands.ReelCutMain.FastStop AND "Unit1.MotionNodes".MotionToPLC.Stauts.ReelCutMain.Done;
   #statTonTimer[811].TON(IN := ("Unit1.Em3.ControlNodes".webGuid.sequence.status.currentStep = #JOB_8_STEP_11) AND "Unit1.Em3.ControlNodes".webGuid.sequence.status.seqActive AND "Unit1.Em3.ControlNodes".webGuid."step".transition[811],
                          PT := #SeqDelayTime);
   IF #statTonTimer[811].Q THEN
       "Unit1.Em3.ControlNodes".webGuid.sequence.status.nextStep := #JOB_8_STEP_91;
   END_IF;
END_REGION

REGION Network 52: Step [891] : JOB[8] Step End
   RUNG wire#powerrail
      { S7_Templates := "SrcType := DInt" } EQ_Contact(in1 := "Unit1.Em3.ControlNodes".webGuid.sequence.status.currentStep, in2 := #JOB_8_STEP_91)
      Contact( "Unit1.Em3.ControlNodes".webGuid.sequence.status.seqActive )
      wire#w1
      Coil( "Unit1.Em3.ControlNodes".webGuid."step".action[891] )
   END_RUNG
   RUNG wire#w1
      Coil( "Unit1.Em3.ControlNodes".webGuid."step".transition[891] )
   END_RUNG
   RUNG wire#w1
      Contact( "Unit1.Em3.ControlNodes".webGuid."step".transition[891] )
      { S7_Templates := "time_type := Time" } #statTonTimer[891].TON(pt := #SeqNoDelayTime, et =>)
      Move(in := #STEP_IDLE, out1 => "Unit1.Em3.ControlNodes".webGuid.sequence.status.nextStep)
   END_RUNG
   // the same network as SCL:
   "Unit1.Em3.ControlNodes".webGuid."step".action[891] := ("Unit1.Em3.ControlNodes".webGuid.sequence.status.currentStep = #JOB_8_STEP_91) AND "Unit1.Em3.ControlNodes".webGuid.sequence.status.seqActive;
   "Unit1.Em3.ControlNodes".webGuid."step".transition[891] := ("Unit1.Em3.ControlNodes".webGuid.sequence.status.currentStep = #JOB_8_STEP_91) AND "Unit1.Em3.ControlNodes".webGuid.sequence.status.seqActive;
   #statTonTimer[891].TON(IN := ("Unit1.Em3.ControlNodes".webGuid.sequence.status.currentStep = #JOB_8_STEP_91) AND "Unit1.Em3.ControlNodes".webGuid.sequence.status.seqActive AND "Unit1.Em3.ControlNodes".webGuid."step".transition[891],
                          PT := #SeqNoDelayTime);
   IF #statTonTimer[891].Q THEN
       "Unit1.Em3.ControlNodes".webGuid.sequence.status.nextStep := #STEP_IDLE;
   END_IF;
END_REGION

REGION Network 53: *************** IMMEDIATE STOP ****************
END_REGION

REGION Network 54: Immediate Stop
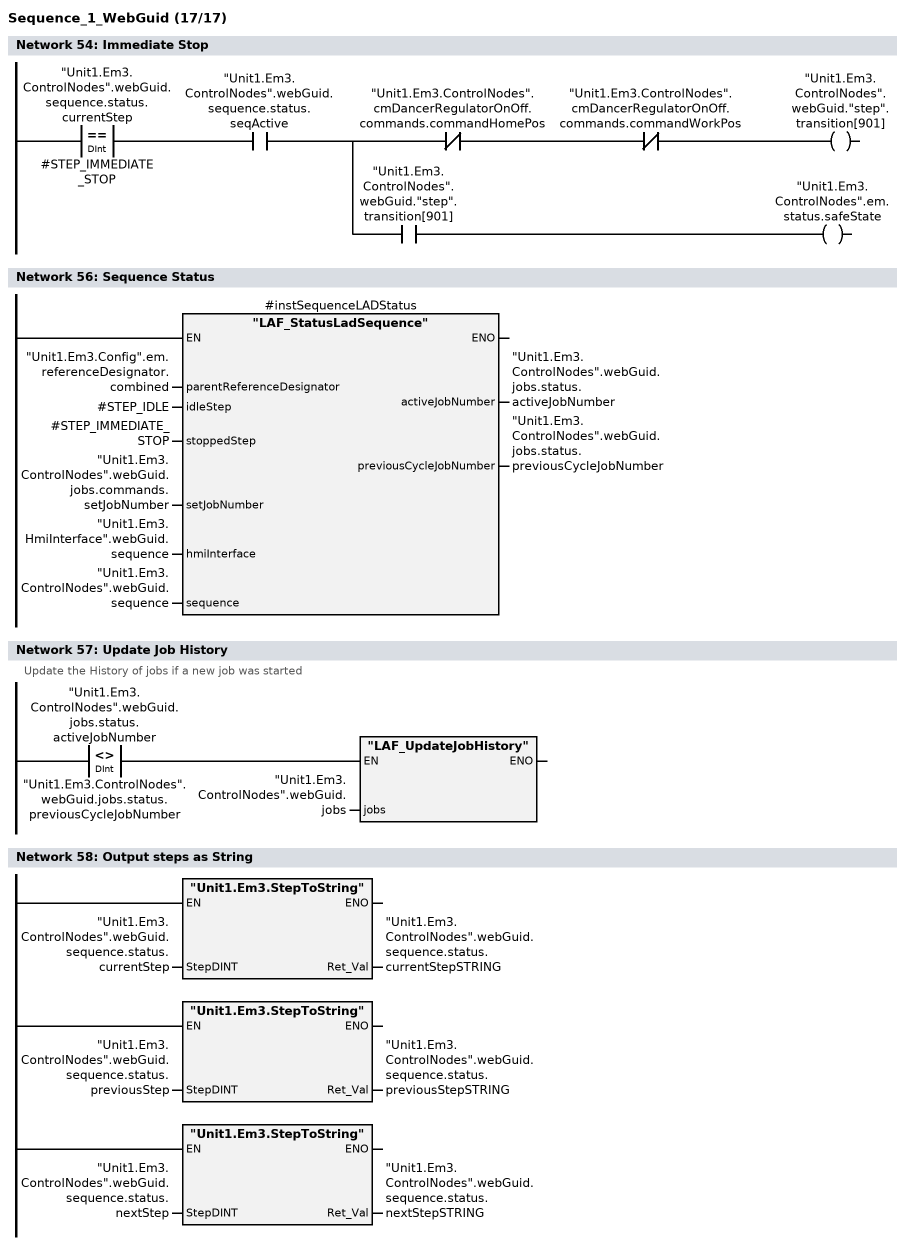
   RUNG wire#powerrail
      { S7_Templates := "SrcType := DInt" } EQ_Contact(in1 := "Unit1.Em3.ControlNodes".webGuid.sequence.status.currentStep, in2 := #STEP_IMMEDIATE_STOP)
      Contact( "Unit1.Em3.ControlNodes".webGuid.sequence.status.seqActive )
      wire#w1
      I_Contact( "Unit1.Em3.ControlNodes".cmDancerRegulatorOnOff.commands.commandHomePos )
      I_Contact( "Unit1.Em3.ControlNodes".cmDancerRegulatorOnOff.commands.commandWorkPos )
      Coil( "Unit1.Em3.ControlNodes".webGuid."step".transition[901] )
   END_RUNG
   RUNG wire#w1
      Contact( "Unit1.Em3.ControlNodes".webGuid."step".transition[901] )
      Coil( "Unit1.Em3.ControlNodes".em.status.safeState )
   END_RUNG
   // the same network as SCL:
   #_w1 := ("Unit1.Em3.ControlNodes".webGuid.sequence.status.currentStep = #STEP_IMMEDIATE_STOP) AND "Unit1.Em3.ControlNodes".webGuid.sequence.status.seqActive;
   "Unit1.Em3.ControlNodes".webGuid."step".transition[901] := #_w1 AND NOT "Unit1.Em3.ControlNodes".cmDancerRegulatorOnOff.commands.commandHomePos AND NOT "Unit1.Em3.ControlNodes".cmDancerRegulatorOnOff.commands.commandWorkPos;
   "Unit1.Em3.ControlNodes".em.status.safeState := #_w1 AND "Unit1.Em3.ControlNodes".webGuid."step".transition[901];
END_REGION

REGION Network 55: *************** STATUS **********************
END_REGION

REGION Network 56: Sequence Status
   RUNG wire#powerrail
      #instSequenceLADStatus(parentReferenceDesignator := "Unit1.Em3.Config".em.referenceDesignator.combined, idleStep := #STEP_IDLE, stoppedStep := #STEP_IMMEDIATE_STOP, setJobNumber := "Unit1.Em3.ControlNodes".webGuid.jobs.commands.setJobNumber, hmiInterface := "Unit1.Em3.HmiInterface".webGuid.sequence, sequence := "Unit1.Em3.ControlNodes".webGuid.sequence, activeJobNumber => "Unit1.Em3.ControlNodes".webGuid.jobs.status.activeJobNumber, previousCycleJobNumber => "Unit1.Em3.ControlNodes".webGuid.jobs.status.previousCycleJobNumber)
   END_RUNG
   // the same network as SCL:
   #instSequenceLADStatus(parentReferenceDesignator := "Unit1.Em3.Config".em.referenceDesignator.combined,   // "LAF_StatusLadSequence"
                          idleStep := #STEP_IDLE,
                          stoppedStep := #STEP_IMMEDIATE_STOP,
                          setJobNumber := "Unit1.Em3.ControlNodes".webGuid.jobs.commands.setJobNumber,
                          hmiInterface := "Unit1.Em3.HmiInterface".webGuid.sequence,
                          sequence := "Unit1.Em3.ControlNodes".webGuid.sequence,
                          activeJobNumber => "Unit1.Em3.ControlNodes".webGuid.jobs.status.activeJobNumber,
                          previousCycleJobNumber => "Unit1.Em3.ControlNodes".webGuid.jobs.status.previousCycleJobNumber);
END_REGION

REGION Network 57: Update Job History
   // Update the History of jobs if a new job was started
   RUNG wire#powerrail
      { S7_Templates := "SrcType := DInt" } NE_Contact(in1 := "Unit1.Em3.ControlNodes".webGuid.jobs.status.activeJobNumber, in2 := "Unit1.Em3.ControlNodes".webGuid.jobs.status.previousCycleJobNumber)
      "LAF_UpdateJobHistory"(jobs := "Unit1.Em3.ControlNodes".webGuid.jobs)
   END_RUNG
   // the same network as SCL:
   IF "Unit1.Em3.ControlNodes".webGuid.jobs.status.activeJobNumber <> "Unit1.Em3.ControlNodes".webGuid.jobs.status.previousCycleJobNumber THEN
       "LAF_UpdateJobHistory"(jobs := "Unit1.Em3.ControlNodes".webGuid.jobs);
   END_IF;
END_REGION

REGION Network 58: Output steps as String
   RUNG wire#powerrail
      "Unit1.Em3.StepToString"(StepDINT := "Unit1.Em3.ControlNodes".webGuid.sequence.status.currentStep, Ret_Val => "Unit1.Em3.ControlNodes".webGuid.sequence.status.currentStepSTRING)
   END_RUNG
   RUNG wire#powerrail
      "Unit1.Em3.StepToString"(StepDINT := "Unit1.Em3.ControlNodes".webGuid.sequence.status.previousStep, Ret_Val => "Unit1.Em3.ControlNodes".webGuid.sequence.status.previousStepSTRING)
   END_RUNG
   RUNG wire#powerrail
      "Unit1.Em3.StepToString"(StepDINT := "Unit1.Em3.ControlNodes".webGuid.sequence.status.nextStep, Ret_Val => "Unit1.Em3.ControlNodes".webGuid.sequence.status.nextStepSTRING)
   END_RUNG
   // the same network as SCL:
   "Unit1.Em3.ControlNodes".webGuid.sequence.status.currentStepSTRING := "Unit1.Em3.StepToString"(StepDINT := "Unit1.Em3.ControlNodes".webGuid.sequence.status.currentStep);
   "Unit1.Em3.ControlNodes".webGuid.sequence.status.previousStepSTRING := "Unit1.Em3.StepToString"(StepDINT := "Unit1.Em3.ControlNodes".webGuid.sequence.status.previousStep);
   "Unit1.Em3.ControlNodes".webGuid.sequence.status.nextStepSTRING := "Unit1.Em3.StepToString"(StepDINT := "Unit1.Em3.ControlNodes".webGuid.sequence.status.nextStep);
END_REGION
END_FUNCTION_BLOCK
